      IF finalPosition == 29 THEN
        ;FOLD SPTP P129 Vel=100 % PDAT1 Tool[1]:SMC Base[0] ;%{PE}
        ;FOLD Parameters ;%{h}
        ;Params IlfProvider=kukaroboter.basistech.inlineforms.movement.spline; Kuka.IsGlobalPoint=False; Kuka.PointName=P129; Kuka.BlendingEnabled=False; Kuka.MoveDataPtpName=PDAT1; Kuka.VelocityPtp=100; Kuka.VelocityFieldEnabled=True; Kuka.ColDetectFieldEnabled=True; Kuka.CurrentCDSetIndex=0; Kuka.MovementParameterFieldEnabled=True; IlfCommand=SPTP
        ;ENDFOLD
        SPTP XP129 WITH $VEL_AXIS[1] = SVEL_JOINT(100.0), $TOOL = STOOL2(FP129), $BASE = SBASE(FP129.BASE_NO), $IPO_MODE = SIPO_MODE(FP129.IPO_FRAME), $LOAD = SLOAD(FP129.TOOL_NO), $ACC_AXIS[1] = SACC_JOINT(PPDAT1), $APO = SAPO_PTP(PPDAT1), $GEAR_JERK[1] = SGEAR_JERK(PPDAT1), $COLLMON_TOL_PRO[1] = USE_CM_PRO_VALUES(0)
        ;ENDFOLD
        ;FOLD SLIN P229 Vel=0.1 m/s CPDAT27 Tool[1]:SMC Base[0] ;%{PE}
        ;FOLD Parameters ;%{h}
        ;Params IlfProvider=kukaroboter.basistech.inlineforms.movement.spline; Kuka.IsGlobalPoint=False; Kuka.PointName=P229; Kuka.BlendingEnabled=False; Kuka.MoveDataName=CPDAT27; Kuka.VelocityPath=0.1; Kuka.VelocityFieldEnabled=True; Kuka.ColDetectFieldEnabled=True; Kuka.CurrentCDSetIndex=0; Kuka.MovementParameterFieldEnabled=True; IlfCommand=SLIN
        ;ENDFOLD
        SLIN XP229 WITH $VEL = SVEL_CP(0.1, , LCPDAT27), $TOOL = STOOL2(FP229), $BASE = SBASE(FP229.BASE_NO), $IPO_MODE = SIPO_MODE(FP229.IPO_FRAME), $LOAD = SLOAD(FP229.TOOL_NO), $ACC = SACC_CP(LCPDAT27), $ORI_TYPE = SORI_TYP(LCPDAT27), $APO = SAPO(LCPDAT27), $JERK = SJERK(LCPDAT27), $COLLMON_TOL_PRO[1] = USE_CM_PRO_VALUES(0)
        ;ENDFOLD
        ;FOLD Gripper SET [1]Gripper1 State=[1]ABIERTA Wait 0.2[s] Check with Strategy 1 ;%{PE}
        ;FOLD Parameters Parameters ;%{h}
        ;Params IlfProvider=GripperTech.GripperSet;setgripper=1;setstate=1;setcont=nocont;waittime=0.2;errorstrategy=1
        ;ENDFOLD
        GRPg_SetStateAndCheck(1, 1, 0.2, 1)
        ;ENDFOLD
        ;FOLD SLIN P129 Vel=0.1 m/s CPDAT28 Tool[1]:SMC Base[0] ;%{PE}
        ;FOLD Parameters ;%{h}
        ;Params IlfProvider=kukaroboter.basistech.inlineforms.movement.spline; Kuka.IsGlobalPoint=False; Kuka.PointName=P129; Kuka.BlendingEnabled=False; Kuka.MoveDataName=CPDAT28; Kuka.VelocityPath=0.1; Kuka.VelocityFieldEnabled=True; Kuka.ColDetectFieldEnabled=True; Kuka.CurrentCDSetIndex=0; Kuka.MovementParameterFieldEnabled=True; IlfCommand=SLIN
        ;ENDFOLD
        SLIN XP129 WITH $VEL = SVEL_CP(0.1, , LCPDAT28), $TOOL = STOOL2(FP129), $BASE = SBASE(FP129.BASE_NO), $IPO_MODE = SIPO_MODE(FP129.IPO_FRAME), $LOAD = SLOAD(FP129.TOOL_NO), $ACC = SACC_CP(LCPDAT28), $ORI_TYPE = SORI_TYP(LCPDAT28), $APO = SAPO(LCPDAT28), $JERK = SJERK(LCPDAT28), $COLLMON_TOL_PRO[1] = USE_CM_PRO_VALUES(0)
        ;ENDFOLD
        ;FOLD SPTP P600 Vel=100 % PDAT1 Tool[1]:SMC Base[0] ;%{PE}
        ;FOLD Parameters ;%{h}
        ;Params IlfProvider=kukaroboter.basistech.inlineforms.movement.spline; Kuka.IsGlobalPoint=False; Kuka.PointName=P600; Kuka.BlendingEnabled=False; Kuka.MoveDataPtpName=PDAT1; Kuka.VelocityPtp=100; Kuka.VelocityFieldEnabled=True; Kuka.ColDetectFieldEnabled=True; Kuka.CurrentCDSetIndex=0; Kuka.MovementParameterFieldEnabled=True; IlfCommand=SPTP
        ;ENDFOLD
        SPTP XP600 WITH $VEL_AXIS[1] = SVEL_JOINT(100.0), $TOOL = STOOL2(FP600), $BASE = SBASE(FP600.BASE_NO), $IPO_MODE = SIPO_MODE(FP600.IPO_FRAME), $LOAD = SLOAD(FP600.TOOL_NO), $ACC_AXIS[1] = SACC_JOINT(PPDAT1), $APO = SAPO_PTP(PPDAT1), $GEAR_JERK[1] = SGEAR_JERK(PPDAT1), $COLLMON_TOL_PRO[1] = USE_CM_PRO_VALUES(0)
        ;ENDFOLD
        ;FOLD SLIN P601 Vel=0.1 m/s CPDAT27 Tool[1]:SMC Base[0] ;%{PE}
        ;FOLD Parameters ;%{h}
        ;Params IlfProvider=kukaroboter.basistech.inlineforms.movement.spline; Kuka.IsGlobalPoint=False; Kuka.PointName=P601; Kuka.BlendingEnabled=False; Kuka.MoveDataName=CPDAT27; Kuka.VelocityPath=0.1; Kuka.VelocityFieldEnabled=True; Kuka.ColDetectFieldEnabled=True; Kuka.CurrentCDSetIndex=0; Kuka.MovementParameterFieldEnabled=True; IlfCommand=SLIN
        ;ENDFOLD
        SLIN XP601 WITH $VEL = SVEL_CP(0.1, , LCPDAT27), $TOOL = STOOL2(FP601), $BASE = SBASE(FP601.BASE_NO), $IPO_MODE = SIPO_MODE(FP601.IPO_FRAME), $LOAD = SLOAD(FP601.TOOL_NO), $ACC = SACC_CP(LCPDAT27), $ORI_TYPE = SORI_TYP(LCPDAT27), $APO = SAPO(LCPDAT27), $JERK = SJERK(LCPDAT27), $COLLMON_TOL_PRO[1] = USE_CM_PRO_VALUES(0)
        ;ENDFOLD
        ;FOLD SLIN P602 Vel=0.1 m/s CPDAT27 Tool[1]:SMC Base[0] ;%{PE}
        ;FOLD Parameters ;%{h}
        ;Params IlfProvider=kukaroboter.basistech.inlineforms.movement.spline; Kuka.IsGlobalPoint=False; Kuka.PointName=P602; Kuka.BlendingEnabled=False; Kuka.MoveDataName=CPDAT27; Kuka.VelocityPath=0.1; Kuka.VelocityFieldEnabled=True; Kuka.ColDetectFieldEnabled=True; Kuka.CurrentCDSetIndex=0; Kuka.MovementParameterFieldEnabled=True; IlfCommand=SLIN
        ;ENDFOLD
        SLIN XP602 WITH $VEL = SVEL_CP(0.1, , LCPDAT27), $TOOL = STOOL2(FP602), $BASE = SBASE(FP602.BASE_NO), $IPO_MODE = SIPO_MODE(FP602.IPO_FRAME), $LOAD = SLOAD(FP602.TOOL_NO), $ACC = SACC_CP(LCPDAT27), $ORI_TYPE = SORI_TYP(LCPDAT27), $APO = SAPO(LCPDAT27), $JERK = SJERK(LCPDAT27), $COLLMON_TOL_PRO[1] = USE_CM_PRO_VALUES(0)
        ;ENDFOLD
      ENDIF

      IF finalPosition == 30 THEN
        ;FOLD SPTP P130 Vel=100 % PDAT1 Tool[1]:SMC Base[0] ;%{PE}
        ;FOLD Parameters ;%{h}
        ;Params IlfProvider=kukaroboter.basistech.inlineforms.movement.spline; Kuka.IsGlobalPoint=False; Kuka.PointName=P130; Kuka.BlendingEnabled=False; Kuka.MoveDataPtpName=PDAT1; Kuka.VelocityPtp=100; Kuka.VelocityFieldEnabled=True; Kuka.ColDetectFieldEnabled=True; Kuka.CurrentCDSetIndex=0; Kuka.MovementParameterFieldEnabled=True; IlfCommand=SPTP
        ;ENDFOLD
        SPTP XP130 WITH $VEL_AXIS[1] = SVEL_JOINT(100.0), $TOOL = STOOL2(FP130), $BASE = SBASE(FP130.BASE_NO), $IPO_MODE = SIPO_MODE(FP130.IPO_FRAME), $LOAD = SLOAD(FP130.TOOL_NO), $ACC_AXIS[1] = SACC_JOINT(PPDAT1), $APO = SAPO_PTP(PPDAT1), $GEAR_JERK[1] = SGEAR_JERK(PPDAT1), $COLLMON_TOL_PRO[1] = USE_CM_PRO_VALUES(0)
        ;ENDFOLD
        ;FOLD SLIN P230 Vel=0.1 m/s CPDAT27 Tool[1]:SMC Base[0] ;%{PE}
        ;FOLD Parameters ;%{h}
        ;Params IlfProvider=kukaroboter.basistech.inlineforms.movement.spline; Kuka.IsGlobalPoint=False; Kuka.PointName=P230; Kuka.BlendingEnabled=False; Kuka.MoveDataName=CPDAT27; Kuka.VelocityPath=0.1; Kuka.VelocityFieldEnabled=True; Kuka.ColDetectFieldEnabled=True; Kuka.CurrentCDSetIndex=0; Kuka.MovementParameterFieldEnabled=True; IlfCommand=SLIN
        ;ENDFOLD
        SLIN XP230 WITH $VEL = SVEL_CP(0.1, , LCPDAT27), $TOOL = STOOL2(FP230), $BASE = SBASE(FP230.BASE_NO), $IPO_MODE = SIPO_MODE(FP230.IPO_FRAME), $LOAD = SLOAD(FP230.TOOL_NO), $ACC = SACC_CP(LCPDAT27), $ORI_TYPE = SORI_TYP(LCPDAT27), $APO = SAPO(LCPDAT27), $JERK = SJERK(LCPDAT27), $COLLMON_TOL_PRO[1] = USE_CM_PRO_VALUES(0)
        ;ENDFOLD
        ;FOLD Gripper SET [1]Gripper1 State=[1]ABIERTA Wait 0.2[s] Check with Strategy 1 ;%{PE}
        ;FOLD Parameters Parameters ;%{h}
        ;Params IlfProvider=GripperTech.GripperSet;setgripper=1;setstate=1;setcont=nocont;waittime=0.2;errorstrategy=1
        ;ENDFOLD
        GRPg_SetStateAndCheck(1, 1, 0.2, 1)
        ;ENDFOLD
        ;FOLD SLIN P130 Vel=0.1 m/s CPDAT28 Tool[1]:SMC Base[0] ;%{PE}
        ;FOLD Parameters ;%{h}
        ;Params IlfProvider=kukaroboter.basistech.inlineforms.movement.spline; Kuka.IsGlobalPoint=False; Kuka.PointName=P130; Kuka.BlendingEnabled=False; Kuka.MoveDataName=CPDAT28; Kuka.VelocityPath=0.1; Kuka.VelocityFieldEnabled=True; Kuka.ColDetectFieldEnabled=True; Kuka.CurrentCDSetIndex=0; Kuka.MovementParameterFieldEnabled=True; IlfCommand=SLIN
        ;ENDFOLD
        SLIN XP130 WITH $VEL = SVEL_CP(0.1, , LCPDAT28), $TOOL = STOOL2(FP130), $BASE = SBASE(FP130.BASE_NO), $IPO_MODE = SIPO_MODE(FP130.IPO_FRAME), $LOAD = SLOAD(FP130.TOOL_NO), $ACC = SACC_CP(LCPDAT28), $ORI_TYPE = SORI_TYP(LCPDAT28), $APO = SAPO(LCPDAT28), $JERK = SJERK(LCPDAT28), $COLLMON_TOL_PRO[1] = USE_CM_PRO_VALUES(0)
        ;ENDFOLD
        ;FOLD SPTP P600 Vel=100 % PDAT1 Tool[1]:SMC Base[0] ;%{PE}
        ;FOLD Parameters ;%{h}
        ;Params IlfProvider=kukaroboter.basistech.inlineforms.movement.spline; Kuka.IsGlobalPoint=False; Kuka.PointName=P600; Kuka.BlendingEnabled=False; Kuka.MoveDataPtpName=PDAT1; Kuka.VelocityPtp=100; Kuka.VelocityFieldEnabled=True; Kuka.ColDetectFieldEnabled=True; Kuka.CurrentCDSetIndex=0; Kuka.MovementParameterFieldEnabled=True; IlfCommand=SPTP
        ;ENDFOLD
        SPTP XP600 WITH $VEL_AXIS[1] = SVEL_JOINT(100.0), $TOOL = STOOL2(FP600), $BASE = SBASE(FP600.BASE_NO), $IPO_MODE = SIPO_MODE(FP600.IPO_FRAME), $LOAD = SLOAD(FP600.TOOL_NO), $ACC_AXIS[1] = SACC_JOINT(PPDAT1), $APO = SAPO_PTP(PPDAT1), $GEAR_JERK[1] = SGEAR_JERK(PPDAT1), $COLLMON_TOL_PRO[1] = USE_CM_PRO_VALUES(0)
        ;ENDFOLD
        ;FOLD SLIN P601 Vel=0.1 m/s CPDAT27 Tool[1]:SMC Base[0] ;%{PE}
        ;FOLD Parameters ;%{h}
        ;Params IlfProvider=kukaroboter.basistech.inlineforms.movement.spline; Kuka.IsGlobalPoint=False; Kuka.PointName=P601; Kuka.BlendingEnabled=False; Kuka.MoveDataName=CPDAT27; Kuka.VelocityPath=0.1; Kuka.VelocityFieldEnabled=True; Kuka.ColDetectFieldEnabled=True; Kuka.CurrentCDSetIndex=0; Kuka.MovementParameterFieldEnabled=True; IlfCommand=SLIN
        ;ENDFOLD
        SLIN XP601 WITH $VEL = SVEL_CP(0.1, , LCPDAT27), $TOOL = STOOL2(FP601), $BASE = SBASE(FP601.BASE_NO), $IPO_MODE = SIPO_MODE(FP601.IPO_FRAME), $LOAD = SLOAD(FP601.TOOL_NO), $ACC = SACC_CP(LCPDAT27), $ORI_TYPE = SORI_TYP(LCPDAT27), $APO = SAPO(LCPDAT27), $JERK = SJERK(LCPDAT27), $COLLMON_TOL_PRO[1] = USE_CM_PRO_VALUES(0)
        ;ENDFOLD
        ;FOLD SLIN P602 Vel=0.1 m/s CPDAT27 Tool[1]:SMC Base[0] ;%{PE}
        ;FOLD Parameters ;%{h}
        ;Params IlfProvider=kukaroboter.basistech.inlineforms.movement.spline; Kuka.IsGlobalPoint=False; Kuka.PointName=P602; Kuka.BlendingEnabled=False; Kuka.MoveDataName=CPDAT27; Kuka.VelocityPath=0.1; Kuka.VelocityFieldEnabled=True; Kuka.ColDetectFieldEnabled=True; Kuka.CurrentCDSetIndex=0; Kuka.MovementParameterFieldEnabled=True; IlfCommand=SLIN
        ;ENDFOLD
        SLIN XP602 WITH $VEL = SVEL_CP(0.1, , LCPDAT27), $TOOL = STOOL2(FP602), $BASE = SBASE(FP602.BASE_NO), $IPO_MODE = SIPO_MODE(FP602.IPO_FRAME), $LOAD = SLOAD(FP602.TOOL_NO), $ACC = SACC_CP(LCPDAT27), $ORI_TYPE = SORI_TYP(LCPDAT27), $APO = SAPO(LCPDAT27), $JERK = SJERK(LCPDAT27), $COLLMON_TOL_PRO[1] = USE_CM_PRO_VALUES(0)
        ;ENDFOLD
      ENDIF

      IF finalPosition == 31 THEN
        ;FOLD SPTP P131 Vel=100 % PDAT1 Tool[1]:SMC Base[0] ;%{PE}
        ;FOLD Parameters ;%{h}
        ;Params IlfProvider=kukaroboter.basistech.inlineforms.movement.spline; Kuka.IsGlobalPoint=False; Kuka.PointName=P131; Kuka.BlendingEnabled=False; Kuka.MoveDataPtpName=PDAT1; Kuka.VelocityPtp=100; Kuka.VelocityFieldEnabled=True; Kuka.ColDetectFieldEnabled=True; Kuka.CurrentCDSetIndex=0; Kuka.MovementParameterFieldEnabled=True; IlfCommand=SPTP
        ;ENDFOLD
        SPTP XP131 WITH $VEL_AXIS[1] = SVEL_JOINT(100.0), $TOOL = STOOL2(FP131), $BASE = SBASE(FP131.BASE_NO), $IPO_MODE = SIPO_MODE(FP131.IPO_FRAME), $LOAD = SLOAD(FP131.TOOL_NO), $ACC_AXIS[1] = SACC_JOINT(PPDAT1), $APO = SAPO_PTP(PPDAT1), $GEAR_JERK[1] = SGEAR_JERK(PPDAT1), $COLLMON_TOL_PRO[1] = USE_CM_PRO_VALUES(0)
        ;ENDFOLD
        ;FOLD SLIN P231 Vel=0.1 m/s CPDAT27 Tool[1]:SMC Base[0] ;%{PE}
        ;FOLD Parameters ;%{h}
        ;Params IlfProvider=kukaroboter.basistech.inlineforms.movement.spline; Kuka.IsGlobalPoint=False; Kuka.PointName=P231; Kuka.BlendingEnabled=False; Kuka.MoveDataName=CPDAT27; Kuka.VelocityPath=0.1; Kuka.VelocityFieldEnabled=True; Kuka.ColDetectFieldEnabled=True; Kuka.CurrentCDSetIndex=0; Kuka.MovementParameterFieldEnabled=True; IlfCommand=SLIN
        ;ENDFOLD
        SLIN XP231 WITH $VEL = SVEL_CP(0.1, , LCPDAT27), $TOOL = STOOL2(FP231), $BASE = SBASE(FP231.BASE_NO), $IPO_MODE = SIPO_MODE(FP231.IPO_FRAME), $LOAD = SLOAD(FP231.TOOL_NO), $ACC = SACC_CP(LCPDAT27), $ORI_TYPE = SORI_TYP(LCPDAT27), $APO = SAPO(LCPDAT27), $JERK = SJERK(LCPDAT27), $COLLMON_TOL_PRO[1] = USE_CM_PRO_VALUES(0)
        ;ENDFOLD
        ;FOLD Gripper SET [1]Gripper1 State=[1]ABIERTA Wait 0.2[s] Check with Strategy 1 ;%{PE}
        ;FOLD Parameters Parameters ;%{h}
        ;Params IlfProvider=GripperTech.GripperSet;setgripper=1;setstate=1;setcont=nocont;waittime=0.2;errorstrategy=1
        ;ENDFOLD
        GRPg_SetStateAndCheck(1, 1, 0.2, 1)
        ;ENDFOLD
        ;FOLD SLIN P131 Vel=0.1 m/s CPDAT28 Tool[1]:SMC Base[0] ;%{PE}
        ;FOLD Parameters ;%{h}
        ;Params IlfProvider=kukaroboter.basistech.inlineforms.movement.spline; Kuka.IsGlobalPoint=False; Kuka.PointName=P131; Kuka.BlendingEnabled=False; Kuka.MoveDataName=CPDAT28; Kuka.VelocityPath=0.1; Kuka.VelocityFieldEnabled=True; Kuka.ColDetectFieldEnabled=True; Kuka.CurrentCDSetIndex=0; Kuka.MovementParameterFieldEnabled=True; IlfCommand=SLIN
        ;ENDFOLD
        SLIN XP131 WITH $VEL = SVEL_CP(0.1, , LCPDAT28), $TOOL = STOOL2(FP131), $BASE = SBASE(FP131.BASE_NO), $IPO_MODE = SIPO_MODE(FP131.IPO_FRAME), $LOAD = SLOAD(FP131.TOOL_NO), $ACC = SACC_CP(LCPDAT28), $ORI_TYPE = SORI_TYP(LCPDAT28), $APO = SAPO(LCPDAT28), $JERK = SJERK(LCPDAT28), $COLLMON_TOL_PRO[1] = USE_CM_PRO_VALUES(0)
        ;ENDFOLD
        ;FOLD SPTP P600 Vel=100 % PDAT1 Tool[1]:SMC Base[0] ;%{PE}
        ;FOLD Parameters ;%{h}
        ;Params IlfProvider=kukaroboter.basistech.inlineforms.movement.spline; Kuka.IsGlobalPoint=False; Kuka.PointName=P600; Kuka.BlendingEnabled=False; Kuka.MoveDataPtpName=PDAT1; Kuka.VelocityPtp=100; Kuka.VelocityFieldEnabled=True; Kuka.ColDetectFieldEnabled=True; Kuka.CurrentCDSetIndex=0; Kuka.MovementParameterFieldEnabled=True; IlfCommand=SPTP
        ;ENDFOLD
        SPTP XP600 WITH $VEL_AXIS[1] = SVEL_JOINT(100.0), $TOOL = STOOL2(FP600), $BASE = SBASE(FP600.BASE_NO), $IPO_MODE = SIPO_MODE(FP600.IPO_FRAME), $LOAD = SLOAD(FP600.TOOL_NO), $ACC_AXIS[1] = SACC_JOINT(PPDAT1), $APO = SAPO_PTP(PPDAT1), $GEAR_JERK[1] = SGEAR_JERK(PPDAT1), $COLLMON_TOL_PRO[1] = USE_CM_PRO_VALUES(0)
        ;ENDFOLD
        ;FOLD SLIN P601 Vel=0.1 m/s CPDAT27 Tool[1]:SMC Base[0] ;%{PE}
        ;FOLD Parameters ;%{h}
        ;Params IlfProvider=kukaroboter.basistech.inlineforms.movement.spline; Kuka.IsGlobalPoint=False; Kuka.PointName=P601; Kuka.BlendingEnabled=False; Kuka.MoveDataName=CPDAT27; Kuka.VelocityPath=0.1; Kuka.VelocityFieldEnabled=True; Kuka.ColDetectFieldEnabled=True; Kuka.CurrentCDSetIndex=0; Kuka.MovementParameterFieldEnabled=True; IlfCommand=SLIN
        ;ENDFOLD
        SLIN XP601 WITH $VEL = SVEL_CP(0.1, , LCPDAT27), $TOOL = STOOL2(FP601), $BASE = SBASE(FP601.BASE_NO), $IPO_MODE = SIPO_MODE(FP601.IPO_FRAME), $LOAD = SLOAD(FP601.TOOL_NO), $ACC = SACC_CP(LCPDAT27), $ORI_TYPE = SORI_TYP(LCPDAT27), $APO = SAPO(LCPDAT27), $JERK = SJERK(LCPDAT27), $COLLMON_TOL_PRO[1] = USE_CM_PRO_VALUES(0)
        ;ENDFOLD
        ;FOLD SLIN P602 Vel=0.1 m/s CPDAT27 Tool[1]:SMC Base[0] ;%{PE}
        ;FOLD Parameters ;%{h}
        ;Params IlfProvider=kukaroboter.basistech.inlineforms.movement.spline; Kuka.IsGlobalPoint=False; Kuka.PointName=P602; Kuka.BlendingEnabled=False; Kuka.MoveDataName=CPDAT27; Kuka.VelocityPath=0.1; Kuka.VelocityFieldEnabled=True; Kuka.ColDetectFieldEnabled=True; Kuka.CurrentCDSetIndex=0; Kuka.MovementParameterFieldEnabled=True; IlfCommand=SLIN
        ;ENDFOLD
        SLIN XP602 WITH $VEL = SVEL_CP(0.1, , LCPDAT27), $TOOL = STOOL2(FP602), $BASE = SBASE(FP602.BASE_NO), $IPO_MODE = SIPO_MODE(FP602.IPO_FRAME), $LOAD = SLOAD(FP602.TOOL_NO), $ACC = SACC_CP(LCPDAT27), $ORI_TYPE = SORI_TYP(LCPDAT27), $APO = SAPO(LCPDAT27), $JERK = SJERK(LCPDAT27), $COLLMON_TOL_PRO[1] = USE_CM_PRO_VALUES(0)
        ;ENDFOLD
      ENDIF

      IF finalPosition == 32 THEN
        ;FOLD SPTP P132 Vel=100 % PDAT1 Tool[1]:SMC Base[0] ;%{PE}
        ;FOLD Parameters ;%{h}
        ;Params IlfProvider=kukaroboter.basistech.inlineforms.movement.spline; Kuka.IsGlobalPoint=False; Kuka.PointName=P132; Kuka.BlendingEnabled=False; Kuka.MoveDataPtpName=PDAT1; Kuka.VelocityPtp=100; Kuka.VelocityFieldEnabled=True; Kuka.ColDetectFieldEnabled=True; Kuka.CurrentCDSetIndex=0; Kuka.MovementParameterFieldEnabled=True; IlfCommand=SPTP
        ;ENDFOLD
        SPTP XP132 WITH $VEL_AXIS[1] = SVEL_JOINT(100.0), $TOOL = STOOL2(FP132), $BASE = SBASE(FP132.BASE_NO), $IPO_MODE = SIPO_MODE(FP132.IPO_FRAME), $LOAD = SLOAD(FP132.TOOL_NO), $ACC_AXIS[1] = SACC_JOINT(PPDAT1), $APO = SAPO_PTP(PPDAT1), $GEAR_JERK[1] = SGEAR_JERK(PPDAT1), $COLLMON_TOL_PRO[1] = USE_CM_PRO_VALUES(0)
        ;ENDFOLD
        ;FOLD SLIN P232 Vel=0.1 m/s CPDAT27 Tool[1]:SMC Base[0] ;%{PE}
        ;FOLD Parameters ;%{h}
        ;Params IlfProvider=kukaroboter.basistech.inlineforms.movement.spline; Kuka.IsGlobalPoint=False; Kuka.PointName=P232; Kuka.BlendingEnabled=False; Kuka.MoveDataName=CPDAT27; Kuka.VelocityPath=0.1; Kuka.VelocityFieldEnabled=True; Kuka.ColDetectFieldEnabled=True; Kuka.CurrentCDSetIndex=0; Kuka.MovementParameterFieldEnabled=True; IlfCommand=SLIN
        ;ENDFOLD
        SLIN XP232 WITH $VEL = SVEL_CP(0.1, , LCPDAT27), $TOOL = STOOL2(FP232), $BASE = SBASE(FP232.BASE_NO), $IPO_MODE = SIPO_MODE(FP232.IPO_FRAME), $LOAD = SLOAD(FP232.TOOL_NO), $ACC = SACC_CP(LCPDAT27), $ORI_TYPE = SORI_TYP(LCPDAT27), $APO = SAPO(LCPDAT27), $JERK = SJERK(LCPDAT27), $COLLMON_TOL_PRO[1] = USE_CM_PRO_VALUES(0)
        ;ENDFOLD
        ;FOLD Gripper SET [1]Gripper1 State=[1]ABIERTA Wait 0.2[s] Check with Strategy 1 ;%{PE}
        ;FOLD Parameters Parameters ;%{h}
        ;Params IlfProvider=GripperTech.GripperSet;setgripper=1;setstate=1;setcont=nocont;waittime=0.2;errorstrategy=1
        ;ENDFOLD
        GRPg_SetStateAndCheck(1, 1, 0.2, 1)
        ;ENDFOLD
        ;FOLD SLIN P132 Vel=0.1 m/s CPDAT28 Tool[1]:SMC Base[0] ;%{PE}
        ;FOLD Parameters ;%{h}
        ;Params IlfProvider=kukaroboter.basistech.inlineforms.movement.spline; Kuka.IsGlobalPoint=False; Kuka.PointName=P132; Kuka.BlendingEnabled=False; Kuka.MoveDataName=CPDAT28; Kuka.VelocityPath=0.1; Kuka.VelocityFieldEnabled=True; Kuka.ColDetectFieldEnabled=True; Kuka.CurrentCDSetIndex=0; Kuka.MovementParameterFieldEnabled=True; IlfCommand=SLIN
        ;ENDFOLD
        SLIN XP132 WITH $VEL = SVEL_CP(0.1, , LCPDAT28), $TOOL = STOOL2(FP132), $BASE = SBASE(FP132.BASE_NO), $IPO_MODE = SIPO_MODE(FP132.IPO_FRAME), $LOAD = SLOAD(FP132.TOOL_NO), $ACC = SACC_CP(LCPDAT28), $ORI_TYPE = SORI_TYP(LCPDAT28), $APO = SAPO(LCPDAT28), $JERK = SJERK(LCPDAT28), $COLLMON_TOL_PRO[1] = USE_CM_PRO_VALUES(0)
        ;ENDFOLD
        ;FOLD SPTP P600 Vel=100 % PDAT1 Tool[1]:SMC Base[0] ;%{PE}
        ;FOLD Parameters ;%{h}
        ;Params IlfProvider=kukaroboter.basistech.inlineforms.movement.spline; Kuka.IsGlobalPoint=False; Kuka.PointName=P600; Kuka.BlendingEnabled=False; Kuka.MoveDataPtpName=PDAT1; Kuka.VelocityPtp=100; Kuka.VelocityFieldEnabled=True; Kuka.ColDetectFieldEnabled=True; Kuka.CurrentCDSetIndex=0; Kuka.MovementParameterFieldEnabled=True; IlfCommand=SPTP
        ;ENDFOLD
        SPTP XP600 WITH $VEL_AXIS[1] = SVEL_JOINT(100.0), $TOOL = STOOL2(FP600), $BASE = SBASE(FP600.BASE_NO), $IPO_MODE = SIPO_MODE(FP600.IPO_FRAME), $LOAD = SLOAD(FP600.TOOL_NO), $ACC_AXIS[1] = SACC_JOINT(PPDAT1), $APO = SAPO_PTP(PPDAT1), $GEAR_JERK[1] = SGEAR_JERK(PPDAT1), $COLLMON_TOL_PRO[1] = USE_CM_PRO_VALUES(0)
        ;ENDFOLD
        ;FOLD SLIN P601 Vel=0.1 m/s CPDAT27 Tool[1]:SMC Base[0] ;%{PE}
        ;FOLD Parameters ;%{h}
        ;Params IlfProvider=kukaroboter.basistech.inlineforms.movement.spline; Kuka.IsGlobalPoint=False; Kuka.PointName=P601; Kuka.BlendingEnabled=False; Kuka.MoveDataName=CPDAT27; Kuka.VelocityPath=0.1; Kuka.VelocityFieldEnabled=True; Kuka.ColDetectFieldEnabled=True; Kuka.CurrentCDSetIndex=0; Kuka.MovementParameterFieldEnabled=True; IlfCommand=SLIN
        ;ENDFOLD
        SLIN XP601 WITH $VEL = SVEL_CP(0.1, , LCPDAT27), $TOOL = STOOL2(FP601), $BASE = SBASE(FP601.BASE_NO), $IPO_MODE = SIPO_MODE(FP601.IPO_FRAME), $LOAD = SLOAD(FP601.TOOL_NO), $ACC = SACC_CP(LCPDAT27), $ORI_TYPE = SORI_TYP(LCPDAT27), $APO = SAPO(LCPDAT27), $JERK = SJERK(LCPDAT27), $COLLMON_TOL_PRO[1] = USE_CM_PRO_VALUES(0)
        ;ENDFOLD
        ;FOLD SLIN P602 Vel=0.1 m/s CPDAT27 Tool[1]:SMC Base[0] ;%{PE}
        ;FOLD Parameters ;%{h}
        ;Params IlfProvider=kukaroboter.basistech.inlineforms.movement.spline; Kuka.IsGlobalPoint=False; Kuka.PointName=P602; Kuka.BlendingEnabled=False; Kuka.MoveDataName=CPDAT27; Kuka.VelocityPath=0.1; Kuka.VelocityFieldEnabled=True; Kuka.ColDetectFieldEnabled=True; Kuka.CurrentCDSetIndex=0; Kuka.MovementParameterFieldEnabled=True; IlfCommand=SLIN
        ;ENDFOLD
        SLIN XP602 WITH $VEL = SVEL_CP(0.1, , LCPDAT27), $TOOL = STOOL2(FP602), $BASE = SBASE(FP602.BASE_NO), $IPO_MODE = SIPO_MODE(FP602.IPO_FRAME), $LOAD = SLOAD(FP602.TOOL_NO), $ACC = SACC_CP(LCPDAT27), $ORI_TYPE = SORI_TYP(LCPDAT27), $APO = SAPO(LCPDAT27), $JERK = SJERK(LCPDAT27), $COLLMON_TOL_PRO[1] = USE_CM_PRO_VALUES(0)
        ;ENDFOLD
      ENDIF

      IF finalPosition == 33 THEN
        ;FOLD SPTP P133 Vel=100 % PDAT1 Tool[1]:SMC Base[0] ;%{PE}
        ;FOLD Parameters ;%{h}
        ;Params IlfProvider=kukaroboter.basistech.inlineforms.movement.spline; Kuka.IsGlobalPoint=False; Kuka.PointName=P133; Kuka.BlendingEnabled=False; Kuka.MoveDataPtpName=PDAT1; Kuka.VelocityPtp=100; Kuka.VelocityFieldEnabled=True; Kuka.ColDetectFieldEnabled=True; Kuka.CurrentCDSetIndex=0; Kuka.MovementParameterFieldEnabled=True; IlfCommand=SPTP
        ;ENDFOLD
        SPTP XP133 WITH $VEL_AXIS[1] = SVEL_JOINT(100.0), $TOOL = STOOL2(FP133), $BASE = SBASE(FP133.BASE_NO), $IPO_MODE = SIPO_MODE(FP133.IPO_FRAME), $LOAD = SLOAD(FP133.TOOL_NO), $ACC_AXIS[1] = SACC_JOINT(PPDAT1), $APO = SAPO_PTP(PPDAT1), $GEAR_JERK[1] = SGEAR_JERK(PPDAT1), $COLLMON_TOL_PRO[1] = USE_CM_PRO_VALUES(0)
        ;ENDFOLD
        ;FOLD SLIN P233 Vel=0.1 m/s CPDAT27 Tool[1]:SMC Base[0] ;%{PE}
        ;FOLD Parameters ;%{h}
        ;Params IlfProvider=kukaroboter.basistech.inlineforms.movement.spline; Kuka.IsGlobalPoint=False; Kuka.PointName=P233; Kuka.BlendingEnabled=False; Kuka.MoveDataName=CPDAT27; Kuka.VelocityPath=0.1; Kuka.VelocityFieldEnabled=True; Kuka.ColDetectFieldEnabled=True; Kuka.CurrentCDSetIndex=0; Kuka.MovementParameterFieldEnabled=True; IlfCommand=SLIN
        ;ENDFOLD
        SLIN XP233 WITH $VEL = SVEL_CP(0.1, , LCPDAT27), $TOOL = STOOL2(FP233), $BASE = SBASE(FP233.BASE_NO), $IPO_MODE = SIPO_MODE(FP233.IPO_FRAME), $LOAD = SLOAD(FP233.TOOL_NO), $ACC = SACC_CP(LCPDAT27), $ORI_TYPE = SORI_TYP(LCPDAT27), $APO = SAPO(LCPDAT27), $JERK = SJERK(LCPDAT27), $COLLMON_TOL_PRO[1] = USE_CM_PRO_VALUES(0)
        ;ENDFOLD
        ;FOLD Gripper SET [1]Gripper1 State=[1]ABIERTA Wait 0.2[s] Check with Strategy 1 ;%{PE}
        ;FOLD Parameters Parameters ;%{h}
        ;Params IlfProvider=GripperTech.GripperSet;setgripper=1;setstate=1;setcont=nocont;waittime=0.2;errorstrategy=1
        ;ENDFOLD
        GRPg_SetStateAndCheck(1, 1, 0.2, 1)
        ;ENDFOLD
        ;FOLD SLIN P133 Vel=0.1 m/s CPDAT28 Tool[1]:SMC Base[0] ;%{PE}
        ;FOLD Parameters ;%{h}
        ;Params IlfProvider=kukaroboter.basistech.inlineforms.movement.spline; Kuka.IsGlobalPoint=False; Kuka.PointName=P133; Kuka.BlendingEnabled=False; Kuka.MoveDataName=CPDAT28; Kuka.VelocityPath=0.1; Kuka.VelocityFieldEnabled=True; Kuka.ColDetectFieldEnabled=True; Kuka.CurrentCDSetIndex=0; Kuka.MovementParameterFieldEnabled=True; IlfCommand=SLIN
        ;ENDFOLD
        SLIN XP133 WITH $VEL = SVEL_CP(0.1, , LCPDAT28), $TOOL = STOOL2(FP133), $BASE = SBASE(FP133.BASE_NO), $IPO_MODE = SIPO_MODE(FP133.IPO_FRAME), $LOAD = SLOAD(FP133.TOOL_NO), $ACC = SACC_CP(LCPDAT28), $ORI_TYPE = SORI_TYP(LCPDAT28), $APO = SAPO(LCPDAT28), $JERK = SJERK(LCPDAT28), $COLLMON_TOL_PRO[1] = USE_CM_PRO_VALUES(0)
        ;ENDFOLD
        ;FOLD SPTP P600 Vel=100 % PDAT1 Tool[1]:SMC Base[0] ;%{PE}
        ;FOLD Parameters ;%{h}
        ;Params IlfProvider=kukaroboter.basistech.inlineforms.movement.spline; Kuka.IsGlobalPoint=False; Kuka.PointName=P600; Kuka.BlendingEnabled=False; Kuka.MoveDataPtpName=PDAT1; Kuka.VelocityPtp=100; Kuka.VelocityFieldEnabled=True; Kuka.ColDetectFieldEnabled=True; Kuka.CurrentCDSetIndex=0; Kuka.MovementParameterFieldEnabled=True; IlfCommand=SPTP
        ;ENDFOLD
        SPTP XP600 WITH $VEL_AXIS[1] = SVEL_JOINT(100.0), $TOOL = STOOL2(FP600), $BASE = SBASE(FP600.BASE_NO), $IPO_MODE = SIPO_MODE(FP600.IPO_FRAME), $LOAD = SLOAD(FP600.TOOL_NO), $ACC_AXIS[1] = SACC_JOINT(PPDAT1), $APO = SAPO_PTP(PPDAT1), $GEAR_JERK[1] = SGEAR_JERK(PPDAT1), $COLLMON_TOL_PRO[1] = USE_CM_PRO_VALUES(0)
        ;ENDFOLD
        ;FOLD SLIN P601 Vel=0.1 m/s CPDAT27 Tool[1]:SMC Base[0] ;%{PE}
        ;FOLD Parameters ;%{h}
        ;Params IlfProvider=kukaroboter.basistech.inlineforms.movement.spline; Kuka.IsGlobalPoint=False; Kuka.PointName=P601; Kuka.BlendingEnabled=False; Kuka.MoveDataName=CPDAT27; Kuka.VelocityPath=0.1; Kuka.VelocityFieldEnabled=True; Kuka.ColDetectFieldEnabled=True; Kuka.CurrentCDSetIndex=0; Kuka.MovementParameterFieldEnabled=True; IlfCommand=SLIN
        ;ENDFOLD
        SLIN XP601 WITH $VEL = SVEL_CP(0.1, , LCPDAT27), $TOOL = STOOL2(FP601), $BASE = SBASE(FP601.BASE_NO), $IPO_MODE = SIPO_MODE(FP601.IPO_FRAME), $LOAD = SLOAD(FP601.TOOL_NO), $ACC = SACC_CP(LCPDAT27), $ORI_TYPE = SORI_TYP(LCPDAT27), $APO = SAPO(LCPDAT27), $JERK = SJERK(LCPDAT27), $COLLMON_TOL_PRO[1] = USE_CM_PRO_VALUES(0)
        ;ENDFOLD
        ;FOLD SLIN P602 Vel=0.1 m/s CPDAT27 Tool[1]:SMC Base[0] ;%{PE}
        ;FOLD Parameters ;%{h}
        ;Params IlfProvider=kukaroboter.basistech.inlineforms.movement.spline; Kuka.IsGlobalPoint=False; Kuka.PointName=P602; Kuka.BlendingEnabled=False; Kuka.MoveDataName=CPDAT27; Kuka.VelocityPath=0.1; Kuka.VelocityFieldEnabled=True; Kuka.ColDetectFieldEnabled=True; Kuka.CurrentCDSetIndex=0; Kuka.MovementParameterFieldEnabled=True; IlfCommand=SLIN
        ;ENDFOLD
        SLIN XP602 WITH $VEL = SVEL_CP(0.1, , LCPDAT27), $TOOL = STOOL2(FP602), $BASE = SBASE(FP602.BASE_NO), $IPO_MODE = SIPO_MODE(FP602.IPO_FRAME), $LOAD = SLOAD(FP602.TOOL_NO), $ACC = SACC_CP(LCPDAT27), $ORI_TYPE = SORI_TYP(LCPDAT27), $APO = SAPO(LCPDAT27), $JERK = SJERK(LCPDAT27), $COLLMON_TOL_PRO[1] = USE_CM_PRO_VALUES(0)
        ;ENDFOLD
      ENDIF

      IF finalPosition == 34 THEN
        ;FOLD SPTP P134 Vel=100 % PDAT1 Tool[1]:SMC Base[0] ;%{PE}
        ;FOLD Parameters ;%{h}
        ;Params IlfProvider=kukaroboter.basistech.inlineforms.movement.spline; Kuka.IsGlobalPoint=False; Kuka.PointName=P134; Kuka.BlendingEnabled=False; Kuka.MoveDataPtpName=PDAT1; Kuka.VelocityPtp=100; Kuka.VelocityFieldEnabled=True; Kuka.ColDetectFieldEnabled=True; Kuka.CurrentCDSetIndex=0; Kuka.MovementParameterFieldEnabled=True; IlfCommand=SPTP
        ;ENDFOLD
        SPTP XP134 WITH $VEL_AXIS[1] = SVEL_JOINT(100.0), $TOOL = STOOL2(FP134), $BASE = SBASE(FP134.BASE_NO), $IPO_MODE = SIPO_MODE(FP134.IPO_FRAME), $LOAD = SLOAD(FP134.TOOL_NO), $ACC_AXIS[1] = SACC_JOINT(PPDAT1), $APO = SAPO_PTP(PPDAT1), $GEAR_JERK[1] = SGEAR_JERK(PPDAT1), $COLLMON_TOL_PRO[1] = USE_CM_PRO_VALUES(0)
        ;ENDFOLD
        ;FOLD SLIN P234 Vel=0.1 m/s CPDAT27 Tool[1]:SMC Base[0] ;%{PE}
        ;FOLD Parameters ;%{h}
        ;Params IlfProvider=kukaroboter.basistech.inlineforms.movement.spline; Kuka.IsGlobalPoint=False; Kuka.PointName=P234; Kuka.BlendingEnabled=False; Kuka.MoveDataName=CPDAT27; Kuka.VelocityPath=0.1; Kuka.VelocityFieldEnabled=True; Kuka.ColDetectFieldEnabled=True; Kuka.CurrentCDSetIndex=0; Kuka.MovementParameterFieldEnabled=True; IlfCommand=SLIN
        ;ENDFOLD
        SLIN XP234 WITH $VEL = SVEL_CP(0.1, , LCPDAT27), $TOOL = STOOL2(FP234), $BASE = SBASE(FP234.BASE_NO), $IPO_MODE = SIPO_MODE(FP234.IPO_FRAME), $LOAD = SLOAD(FP234.TOOL_NO), $ACC = SACC_CP(LCPDAT27), $ORI_TYPE = SORI_TYP(LCPDAT27), $APO = SAPO(LCPDAT27), $JERK = SJERK(LCPDAT27), $COLLMON_TOL_PRO[1] = USE_CM_PRO_VALUES(0)
        ;ENDFOLD
        ;FOLD Gripper SET [1]Gripper1 State=[1]ABIERTA Wait 0.2[s] Check with Strategy 1 ;%{PE}
        ;FOLD Parameters Parameters ;%{h}
        ;Params IlfProvider=GripperTech.GripperSet;setgripper=1;setstate=1;setcont=nocont;waittime=0.2;errorstrategy=1
        ;ENDFOLD
        GRPg_SetStateAndCheck(1, 1, 0.2, 1)
        ;ENDFOLD
        ;FOLD SLIN P134 Vel=0.1 m/s CPDAT28 Tool[1]:SMC Base[0] ;%{PE}
        ;FOLD Parameters ;%{h}
        ;Params IlfProvider=kukaroboter.basistech.inlineforms.movement.spline; Kuka.IsGlobalPoint=False; Kuka.PointName=P134; Kuka.BlendingEnabled=False; Kuka.MoveDataName=CPDAT28; Kuka.VelocityPath=0.1; Kuka.VelocityFieldEnabled=True; Kuka.ColDetectFieldEnabled=True; Kuka.CurrentCDSetIndex=0; Kuka.MovementParameterFieldEnabled=True; IlfCommand=SLIN
        ;ENDFOLD
        SLIN XP134 WITH $VEL = SVEL_CP(0.1, , LCPDAT28), $TOOL = STOOL2(FP134), $BASE = SBASE(FP134.BASE_NO), $IPO_MODE = SIPO_MODE(FP134.IPO_FRAME), $LOAD = SLOAD(FP134.TOOL_NO), $ACC = SACC_CP(LCPDAT28), $ORI_TYPE = SORI_TYP(LCPDAT28), $APO = SAPO(LCPDAT28), $JERK = SJERK(LCPDAT28), $COLLMON_TOL_PRO[1] = USE_CM_PRO_VALUES(0)
        ;ENDFOLD
        ;FOLD SPTP P600 Vel=100 % PDAT1 Tool[1]:SMC Base[0] ;%{PE}
        ;FOLD Parameters ;%{h}
        ;Params IlfProvider=kukaroboter.basistech.inlineforms.movement.spline; Kuka.IsGlobalPoint=False; Kuka.PointName=P600; Kuka.BlendingEnabled=False; Kuka.MoveDataPtpName=PDAT1; Kuka.VelocityPtp=100; Kuka.VelocityFieldEnabled=True; Kuka.ColDetectFieldEnabled=True; Kuka.CurrentCDSetIndex=0; Kuka.MovementParameterFieldEnabled=True; IlfCommand=SPTP
        ;ENDFOLD
        SPTP XP600 WITH $VEL_AXIS[1] = SVEL_JOINT(100.0), $TOOL = STOOL2(FP600), $BASE = SBASE(FP600.BASE_NO), $IPO_MODE = SIPO_MODE(FP600.IPO_FRAME), $LOAD = SLOAD(FP600.TOOL_NO), $ACC_AXIS[1] = SACC_JOINT(PPDAT1), $APO = SAPO_PTP(PPDAT1), $GEAR_JERK[1] = SGEAR_JERK(PPDAT1), $COLLMON_TOL_PRO[1] = USE_CM_PRO_VALUES(0)
        ;ENDFOLD
        ;FOLD SLIN P601 Vel=0.1 m/s CPDAT27 Tool[1]:SMC Base[0] ;%{PE}
        ;FOLD Parameters ;%{h}
        ;Params IlfProvider=kukaroboter.basistech.inlineforms.movement.spline; Kuka.IsGlobalPoint=False; Kuka.PointName=P601; Kuka.BlendingEnabled=False; Kuka.MoveDataName=CPDAT27; Kuka.VelocityPath=0.1; Kuka.VelocityFieldEnabled=True; Kuka.ColDetectFieldEnabled=True; Kuka.CurrentCDSetIndex=0; Kuka.MovementParameterFieldEnabled=True; IlfCommand=SLIN
        ;ENDFOLD
        SLIN XP601 WITH $VEL = SVEL_CP(0.1, , LCPDAT27), $TOOL = STOOL2(FP601), $BASE = SBASE(FP601.BASE_NO), $IPO_MODE = SIPO_MODE(FP601.IPO_FRAME), $LOAD = SLOAD(FP601.TOOL_NO), $ACC = SACC_CP(LCPDAT27), $ORI_TYPE = SORI_TYP(LCPDAT27), $APO = SAPO(LCPDAT27), $JERK = SJERK(LCPDAT27), $COLLMON_TOL_PRO[1] = USE_CM_PRO_VALUES(0)
        ;ENDFOLD
        ;FOLD SLIN P602 Vel=0.1 m/s CPDAT27 Tool[1]:SMC Base[0] ;%{PE}
        ;FOLD Parameters ;%{h}
        ;Params IlfProvider=kukaroboter.basistech.inlineforms.movement.spline; Kuka.IsGlobalPoint=False; Kuka.PointName=P602; Kuka.BlendingEnabled=False; Kuka.MoveDataName=CPDAT27; Kuka.VelocityPath=0.1; Kuka.VelocityFieldEnabled=True; Kuka.ColDetectFieldEnabled=True; Kuka.CurrentCDSetIndex=0; Kuka.MovementParameterFieldEnabled=True; IlfCommand=SLIN
        ;ENDFOLD
        SLIN XP602 WITH $VEL = SVEL_CP(0.1, , LCPDAT27), $TOOL = STOOL2(FP602), $BASE = SBASE(FP602.BASE_NO), $IPO_MODE = SIPO_MODE(FP602.IPO_FRAME), $LOAD = SLOAD(FP602.TOOL_NO), $ACC = SACC_CP(LCPDAT27), $ORI_TYPE = SORI_TYP(LCPDAT27), $APO = SAPO(LCPDAT27), $JERK = SJERK(LCPDAT27), $COLLMON_TOL_PRO[1] = USE_CM_PRO_VALUES(0)
        ;ENDFOLD
      ENDIF

      IF finalPosition == 35 THEN
        ;FOLD SPTP P135 Vel=100 % PDAT1 Tool[1]:SMC Base[0] ;%{PE}
        ;FOLD Parameters ;%{h}
        ;Params IlfProvider=kukaroboter.basistech.inlineforms.movement.spline; Kuka.IsGlobalPoint=False; Kuka.PointName=P135; Kuka.BlendingEnabled=False; Kuka.MoveDataPtpName=PDAT1; Kuka.VelocityPtp=100; Kuka.VelocityFieldEnabled=True; Kuka.ColDetectFieldEnabled=True; Kuka.CurrentCDSetIndex=0; Kuka.MovementParameterFieldEnabled=True; IlfCommand=SPTP
        ;ENDFOLD
        SPTP XP135 WITH $VEL_AXIS[1] = SVEL_JOINT(100.0), $TOOL = STOOL2(FP135), $BASE = SBASE(FP135.BASE_NO), $IPO_MODE = SIPO_MODE(FP135.IPO_FRAME), $LOAD = SLOAD(FP135.TOOL_NO), $ACC_AXIS[1] = SACC_JOINT(PPDAT1), $APO = SAPO_PTP(PPDAT1), $GEAR_JERK[1] = SGEAR_JERK(PPDAT1), $COLLMON_TOL_PRO[1] = USE_CM_PRO_VALUES(0)
        ;ENDFOLD
        ;FOLD SLIN P235 Vel=0.1 m/s CPDAT27 Tool[1]:SMC Base[0] ;%{PE}
        ;FOLD Parameters ;%{h}
        ;Params IlfProvider=kukaroboter.basistech.inlineforms.movement.spline; Kuka.IsGlobalPoint=False; Kuka.PointName=P235; Kuka.BlendingEnabled=False; Kuka.MoveDataName=CPDAT27; Kuka.VelocityPath=0.1; Kuka.VelocityFieldEnabled=True; Kuka.ColDetectFieldEnabled=True; Kuka.CurrentCDSetIndex=0; Kuka.MovementParameterFieldEnabled=True; IlfCommand=SLIN
        ;ENDFOLD
        SLIN XP235 WITH $VEL = SVEL_CP(0.1, , LCPDAT27), $TOOL = STOOL2(FP235), $BASE = SBASE(FP235.BASE_NO), $IPO_MODE = SIPO_MODE(FP235.IPO_FRAME), $LOAD = SLOAD(FP235.TOOL_NO), $ACC = SACC_CP(LCPDAT27), $ORI_TYPE = SORI_TYP(LCPDAT27), $APO = SAPO(LCPDAT27), $JERK = SJERK(LCPDAT27), $COLLMON_TOL_PRO[1] = USE_CM_PRO_VALUES(0)
        ;ENDFOLD
        ;FOLD Gripper SET [1]Gripper1 State=[1]ABIERTA Wait 0.2[s] Check with Strategy 1 ;%{PE}
        ;FOLD Parameters Parameters ;%{h}
        ;Params IlfProvider=GripperTech.GripperSet;setgripper=1;setstate=1;setcont=nocont;waittime=0.2;errorstrategy=1
        ;ENDFOLD
        GRPg_SetStateAndCheck(1, 1, 0.2, 1)
        ;ENDFOLD
        ;FOLD SLIN P135 Vel=0.1 m/s CPDAT28 Tool[1]:SMC Base[0] ;%{PE}
        ;FOLD Parameters ;%{h}
        ;Params IlfProvider=kukaroboter.basistech.inlineforms.movement.spline; Kuka.IsGlobalPoint=False; Kuka.PointName=P135; Kuka.BlendingEnabled=False; Kuka.MoveDataName=CPDAT28; Kuka.VelocityPath=0.1; Kuka.VelocityFieldEnabled=True; Kuka.ColDetectFieldEnabled=True; Kuka.CurrentCDSetIndex=0; Kuka.MovementParameterFieldEnabled=True; IlfCommand=SLIN
        ;ENDFOLD
        SLIN XP135 WITH $VEL = SVEL_CP(0.1, , LCPDAT28), $TOOL = STOOL2(FP135), $BASE = SBASE(FP135.BASE_NO), $IPO_MODE = SIPO_MODE(FP135.IPO_FRAME), $LOAD = SLOAD(FP135.TOOL_NO), $ACC = SACC_CP(LCPDAT28), $ORI_TYPE = SORI_TYP(LCPDAT28), $APO = SAPO(LCPDAT28), $JERK = SJERK(LCPDAT28), $COLLMON_TOL_PRO[1] = USE_CM_PRO_VALUES(0)
        ;ENDFOLD
        ;FOLD SPTP P600 Vel=100 % PDAT1 Tool[1]:SMC Base[0] ;%{PE}
        ;FOLD Parameters ;%{h}
        ;Params IlfProvider=kukaroboter.basistech.inlineforms.movement.spline; Kuka.IsGlobalPoint=False; Kuka.PointName=P600; Kuka.BlendingEnabled=False; Kuka.MoveDataPtpName=PDAT1; Kuka.VelocityPtp=100; Kuka.VelocityFieldEnabled=True; Kuka.ColDetectFieldEnabled=True; Kuka.CurrentCDSetIndex=0; Kuka.MovementParameterFieldEnabled=True; IlfCommand=SPTP
        ;ENDFOLD
        SPTP XP600 WITH $VEL_AXIS[1] = SVEL_JOINT(100.0), $TOOL = STOOL2(FP600), $BASE = SBASE(FP600.BASE_NO), $IPO_MODE = SIPO_MODE(FP600.IPO_FRAME), $LOAD = SLOAD(FP600.TOOL_NO), $ACC_AXIS[1] = SACC_JOINT(PPDAT1), $APO = SAPO_PTP(PPDAT1), $GEAR_JERK[1] = SGEAR_JERK(PPDAT1), $COLLMON_TOL_PRO[1] = USE_CM_PRO_VALUES(0)
        ;ENDFOLD
        ;FOLD SLIN P601 Vel=0.1 m/s CPDAT27 Tool[1]:SMC Base[0] ;%{PE}
        ;FOLD Parameters ;%{h}
        ;Params IlfProvider=kukaroboter.basistech.inlineforms.movement.spline; Kuka.IsGlobalPoint=False; Kuka.PointName=P601; Kuka.BlendingEnabled=False; Kuka.MoveDataName=CPDAT27; Kuka.VelocityPath=0.1; Kuka.VelocityFieldEnabled=True; Kuka.ColDetectFieldEnabled=True; Kuka.CurrentCDSetIndex=0; Kuka.MovementParameterFieldEnabled=True; IlfCommand=SLIN
        ;ENDFOLD
        SLIN XP601 WITH $VEL = SVEL_CP(0.1, , LCPDAT27), $TOOL = STOOL2(FP601), $BASE = SBASE(FP601.BASE_NO), $IPO_MODE = SIPO_MODE(FP601.IPO_FRAME), $LOAD = SLOAD(FP601.TOOL_NO), $ACC = SACC_CP(LCPDAT27), $ORI_TYPE = SORI_TYP(LCPDAT27), $APO = SAPO(LCPDAT27), $JERK = SJERK(LCPDAT27), $COLLMON_TOL_PRO[1] = USE_CM_PRO_VALUES(0)
        ;ENDFOLD
        ;FOLD SLIN P602 Vel=0.1 m/s CPDAT27 Tool[1]:SMC Base[0] ;%{PE}
        ;FOLD Parameters ;%{h}
        ;Params IlfProvider=kukaroboter.basistech.inlineforms.movement.spline; Kuka.IsGlobalPoint=False; Kuka.PointName=P602; Kuka.BlendingEnabled=False; Kuka.MoveDataName=CPDAT27; Kuka.VelocityPath=0.1; Kuka.VelocityFieldEnabled=True; Kuka.ColDetectFieldEnabled=True; Kuka.CurrentCDSetIndex=0; Kuka.MovementParameterFieldEnabled=True; IlfCommand=SLIN
        ;ENDFOLD
        SLIN XP602 WITH $VEL = SVEL_CP(0.1, , LCPDAT27), $TOOL = STOOL2(FP602), $BASE = SBASE(FP602.BASE_NO), $IPO_MODE = SIPO_MODE(FP602.IPO_FRAME), $LOAD = SLOAD(FP602.TOOL_NO), $ACC = SACC_CP(LCPDAT27), $ORI_TYPE = SORI_TYP(LCPDAT27), $APO = SAPO(LCPDAT27), $JERK = SJERK(LCPDAT27), $COLLMON_TOL_PRO[1] = USE_CM_PRO_VALUES(0)
        ;ENDFOLD
      ENDIF

      IF finalPosition == 36 THEN
        ;FOLD SPTP P136 Vel=100 % PDAT1 Tool[1]:SMC Base[0] ;%{PE}
        ;FOLD Parameters ;%{h}
        ;Params IlfProvider=kukaroboter.basistech.inlineforms.movement.spline; Kuka.IsGlobalPoint=False; Kuka.PointName=P136; Kuka.BlendingEnabled=False; Kuka.MoveDataPtpName=PDAT1; Kuka.VelocityPtp=100; Kuka.VelocityFieldEnabled=True; Kuka.ColDetectFieldEnabled=True; Kuka.CurrentCDSetIndex=0; Kuka.MovementParameterFieldEnabled=True; IlfCommand=SPTP
        ;ENDFOLD
        SPTP XP136 WITH $VEL_AXIS[1] = SVEL_JOINT(100.0), $TOOL = STOOL2(FP136), $BASE = SBASE(FP136.BASE_NO), $IPO_MODE = SIPO_MODE(FP136.IPO_FRAME), $LOAD = SLOAD(FP136.TOOL_NO), $ACC_AXIS[1] = SACC_JOINT(PPDAT1), $APO = SAPO_PTP(PPDAT1), $GEAR_JERK[1] = SGEAR_JERK(PPDAT1), $COLLMON_TOL_PRO[1] = USE_CM_PRO_VALUES(0)
        ;ENDFOLD
        ;FOLD SLIN P236 Vel=0.1 m/s CPDAT27 Tool[1]:SMC Base[0] ;%{PE}
        ;FOLD Parameters ;%{h}
        ;Params IlfProvider=kukaroboter.basistech.inlineforms.movement.spline; Kuka.IsGlobalPoint=False; Kuka.PointName=P236; Kuka.BlendingEnabled=False; Kuka.MoveDataName=CPDAT27; Kuka.VelocityPath=0.1; Kuka.VelocityFieldEnabled=True; Kuka.ColDetectFieldEnabled=True; Kuka.CurrentCDSetIndex=0; Kuka.MovementParameterFieldEnabled=True; IlfCommand=SLIN
        ;ENDFOLD
        SLIN XP236 WITH $VEL = SVEL_CP(0.1, , LCPDAT27), $TOOL = STOOL2(FP236), $BASE = SBASE(FP236.BASE_NO), $IPO_MODE = SIPO_MODE(FP236.IPO_FRAME), $LOAD = SLOAD(FP236.TOOL_NO), $ACC = SACC_CP(LCPDAT27), $ORI_TYPE = SORI_TYP(LCPDAT27), $APO = SAPO(LCPDAT27), $JERK = SJERK(LCPDAT27), $COLLMON_TOL_PRO[1] = USE_CM_PRO_VALUES(0)
        ;ENDFOLD
        ;FOLD Gripper SET [1]Gripper1 State=[1]ABIERTA Wait 0.2[s] Check with Strategy 1 ;%{PE}
        ;FOLD Parameters Parameters ;%{h}
        ;Params IlfProvider=GripperTech.GripperSet;setgripper=1;setstate=1;setcont=nocont;waittime=0.2;errorstrategy=1
        ;ENDFOLD
        GRPg_SetStateAndCheck(1, 1, 0.2, 1)
        ;ENDFOLD
        ;FOLD SLIN P136 Vel=0.1 m/s CPDAT28 Tool[1]:SMC Base[0] ;%{PE}
        ;FOLD Parameters ;%{h}
        ;Params IlfProvider=kukaroboter.basistech.inlineforms.movement.spline; Kuka.IsGlobalPoint=False; Kuka.PointName=P136; Kuka.BlendingEnabled=False; Kuka.MoveDataName=CPDAT28; Kuka.VelocityPath=0.1; Kuka.VelocityFieldEnabled=True; Kuka.ColDetectFieldEnabled=True; Kuka.CurrentCDSetIndex=0; Kuka.MovementParameterFieldEnabled=True; IlfCommand=SLIN
        ;ENDFOLD
        SLIN XP136 WITH $VEL = SVEL_CP(0.1, , LCPDAT28), $TOOL = STOOL2(FP136), $BASE = SBASE(FP136.BASE_NO), $IPO_MODE = SIPO_MODE(FP136.IPO_FRAME), $LOAD = SLOAD(FP136.TOOL_NO), $ACC = SACC_CP(LCPDAT28), $ORI_TYPE = SORI_TYP(LCPDAT28), $APO = SAPO(LCPDAT28), $JERK = SJERK(LCPDAT28), $COLLMON_TOL_PRO[1] = USE_CM_PRO_VALUES(0)
        ;ENDFOLD
        ;FOLD SPTP P600 Vel=100 % PDAT1 Tool[1]:SMC Base[0] ;%{PE}
        ;FOLD Parameters ;%{h}
        ;Params IlfProvider=kukaroboter.basistech.inlineforms.movement.spline; Kuka.IsGlobalPoint=False; Kuka.PointName=P600; Kuka.BlendingEnabled=False; Kuka.MoveDataPtpName=PDAT1; Kuka.VelocityPtp=100; Kuka.VelocityFieldEnabled=True; Kuka.ColDetectFieldEnabled=True; Kuka.CurrentCDSetIndex=0; Kuka.MovementParameterFieldEnabled=True; IlfCommand=SPTP
        ;ENDFOLD
        SPTP XP600 WITH $VEL_AXIS[1] = SVEL_JOINT(100.0), $TOOL = STOOL2(FP600), $BASE = SBASE(FP600.BASE_NO), $IPO_MODE = SIPO_MODE(FP600.IPO_FRAME), $LOAD = SLOAD(FP600.TOOL_NO), $ACC_AXIS[1] = SACC_JOINT(PPDAT1), $APO = SAPO_PTP(PPDAT1), $GEAR_JERK[1] = SGEAR_JERK(PPDAT1), $COLLMON_TOL_PRO[1] = USE_CM_PRO_VALUES(0)
        ;ENDFOLD
        ;FOLD SLIN P601 Vel=0.1 m/s CPDAT27 Tool[1]:SMC Base[0] ;%{PE}
        ;FOLD Parameters ;%{h}
        ;Params IlfProvider=kukaroboter.basistech.inlineforms.movement.spline; Kuka.IsGlobalPoint=False; Kuka.PointName=P601; Kuka.BlendingEnabled=False; Kuka.MoveDataName=CPDAT27; Kuka.VelocityPath=0.1; Kuka.VelocityFieldEnabled=True; Kuka.ColDetectFieldEnabled=True; Kuka.CurrentCDSetIndex=0; Kuka.MovementParameterFieldEnabled=True; IlfCommand=SLIN
        ;ENDFOLD
        SLIN XP601 WITH $VEL = SVEL_CP(0.1, , LCPDAT27), $TOOL = STOOL2(FP601), $BASE = SBASE(FP601.BASE_NO), $IPO_MODE = SIPO_MODE(FP601.IPO_FRAME), $LOAD = SLOAD(FP601.TOOL_NO), $ACC = SACC_CP(LCPDAT27), $ORI_TYPE = SORI_TYP(LCPDAT27), $APO = SAPO(LCPDAT27), $JERK = SJERK(LCPDAT27), $COLLMON_TOL_PRO[1] = USE_CM_PRO_VALUES(0)
        ;ENDFOLD
        ;FOLD SLIN P602 Vel=0.1 m/s CPDAT27 Tool[1]:SMC Base[0] ;%{PE}
        ;FOLD Parameters ;%{h}
        ;Params IlfProvider=kukaroboter.basistech.inlineforms.movement.spline; Kuka.IsGlobalPoint=False; Kuka.PointName=P602; Kuka.BlendingEnabled=False; Kuka.MoveDataName=CPDAT27; Kuka.VelocityPath=0.1; Kuka.VelocityFieldEnabled=True; Kuka.ColDetectFieldEnabled=True; Kuka.CurrentCDSetIndex=0; Kuka.MovementParameterFieldEnabled=True; IlfCommand=SLIN
        ;ENDFOLD
        SLIN XP602 WITH $VEL = SVEL_CP(0.1, , LCPDAT27), $TOOL = STOOL2(FP602), $BASE = SBASE(FP602.BASE_NO), $IPO_MODE = SIPO_MODE(FP602.IPO_FRAME), $LOAD = SLOAD(FP602.TOOL_NO), $ACC = SACC_CP(LCPDAT27), $ORI_TYPE = SORI_TYP(LCPDAT27), $APO = SAPO(LCPDAT27), $JERK = SJERK(LCPDAT27), $COLLMON_TOL_PRO[1] = USE_CM_PRO_VALUES(0)
        ;ENDFOLD
      ENDIF

      IF finalPosition == 37 THEN
        ;FOLD SPTP P137 Vel=100 % PDAT1 Tool[1]:SMC Base[0] ;%{PE}
        ;FOLD Parameters ;%{h}
        ;Params IlfProvider=kukaroboter.basistech.inlineforms.movement.spline; Kuka.IsGlobalPoint=False; Kuka.PointName=P137; Kuka.BlendingEnabled=False; Kuka.MoveDataPtpName=PDAT1; Kuka.VelocityPtp=100; Kuka.VelocityFieldEnabled=True; Kuka.ColDetectFieldEnabled=True; Kuka.CurrentCDSetIndex=0; Kuka.MovementParameterFieldEnabled=True; IlfCommand=SPTP
        ;ENDFOLD
        SPTP XP137 WITH $VEL_AXIS[1] = SVEL_JOINT(100.0), $TOOL = STOOL2(FP137), $BASE = SBASE(FP137.BASE_NO), $IPO_MODE = SIPO_MODE(FP137.IPO_FRAME), $LOAD = SLOAD(FP137.TOOL_NO), $ACC_AXIS[1] = SACC_JOINT(PPDAT1), $APO = SAPO_PTP(PPDAT1), $GEAR_JERK[1] = SGEAR_JERK(PPDAT1), $COLLMON_TOL_PRO[1] = USE_CM_PRO_VALUES(0)
        ;ENDFOLD
        ;FOLD SLIN P237 Vel=0.1 m/s CPDAT27 Tool[1]:SMC Base[0] ;%{PE}
        ;FOLD Parameters ;%{h}
        ;Params IlfProvider=kukaroboter.basistech.inlineforms.movement.spline; Kuka.IsGlobalPoint=False; Kuka.PointName=P237; Kuka.BlendingEnabled=False; Kuka.MoveDataName=CPDAT27; Kuka.VelocityPath=0.1; Kuka.VelocityFieldEnabled=True; Kuka.ColDetectFieldEnabled=True; Kuka.CurrentCDSetIndex=0; Kuka.MovementParameterFieldEnabled=True; IlfCommand=SLIN
        ;ENDFOLD
        SLIN XP237 WITH $VEL = SVEL_CP(0.1, , LCPDAT27), $TOOL = STOOL2(FP237), $BASE = SBASE(FP237.BASE_NO), $IPO_MODE = SIPO_MODE(FP237.IPO_FRAME), $LOAD = SLOAD(FP237.TOOL_NO), $ACC = SACC_CP(LCPDAT27), $ORI_TYPE = SORI_TYP(LCPDAT27), $APO = SAPO(LCPDAT27), $JERK = SJERK(LCPDAT27), $COLLMON_TOL_PRO[1] = USE_CM_PRO_VALUES(0)
        ;ENDFOLD
        ;FOLD Gripper SET [1]Gripper1 State=[1]ABIERTA Wait 0.2[s] Check with Strategy 1 ;%{PE}
        ;FOLD Parameters Parameters ;%{h}
        ;Params IlfProvider=GripperTech.GripperSet;setgripper=1;setstate=1;setcont=nocont;waittime=0.2;errorstrategy=1
        ;ENDFOLD
        GRPg_SetStateAndCheck(1, 1, 0.2, 1)
        ;ENDFOLD
        ;FOLD SLIN P137 Vel=0.1 m/s CPDAT28 Tool[1]:SMC Base[0] ;%{PE}
        ;FOLD Parameters ;%{h}
        ;Params IlfProvider=kukaroboter.basistech.inlineforms.movement.spline; Kuka.IsGlobalPoint=False; Kuka.PointName=P137; Kuka.BlendingEnabled=False; Kuka.MoveDataName=CPDAT28; Kuka.VelocityPath=0.1; Kuka.VelocityFieldEnabled=True; Kuka.ColDetectFieldEnabled=True; Kuka.CurrentCDSetIndex=0; Kuka.MovementParameterFieldEnabled=True; IlfCommand=SLIN
        ;ENDFOLD
        SLIN XP137 WITH $VEL = SVEL_CP(0.1, , LCPDAT28), $TOOL = STOOL2(FP137), $BASE = SBASE(FP137.BASE_NO), $IPO_MODE = SIPO_MODE(FP137.IPO_FRAME), $LOAD = SLOAD(FP137.TOOL_NO), $ACC = SACC_CP(LCPDAT28), $ORI_TYPE = SORI_TYP(LCPDAT28), $APO = SAPO(LCPDAT28), $JERK = SJERK(LCPDAT28), $COLLMON_TOL_PRO[1] = USE_CM_PRO_VALUES(0)
        ;ENDFOLD
        ;FOLD SPTP P600 Vel=100 % PDAT1 Tool[1]:SMC Base[0] ;%{PE}
        ;FOLD Parameters ;%{h}
        ;Params IlfProvider=kukaroboter.basistech.inlineforms.movement.spline; Kuka.IsGlobalPoint=False; Kuka.PointName=P600; Kuka.BlendingEnabled=False; Kuka.MoveDataPtpName=PDAT1; Kuka.VelocityPtp=100; Kuka.VelocityFieldEnabled=True; Kuka.ColDetectFieldEnabled=True; Kuka.CurrentCDSetIndex=0; Kuka.MovementParameterFieldEnabled=True; IlfCommand=SPTP
        ;ENDFOLD
        SPTP XP600 WITH $VEL_AXIS[1] = SVEL_JOINT(100.0), $TOOL = STOOL2(FP600), $BASE = SBASE(FP600.BASE_NO), $IPO_MODE = SIPO_MODE(FP600.IPO_FRAME), $LOAD = SLOAD(FP600.TOOL_NO), $ACC_AXIS[1] = SACC_JOINT(PPDAT1), $APO = SAPO_PTP(PPDAT1), $GEAR_JERK[1] = SGEAR_JERK(PPDAT1), $COLLMON_TOL_PRO[1] = USE_CM_PRO_VALUES(0)
        ;ENDFOLD
        ;FOLD SLIN P601 Vel=0.1 m/s CPDAT27 Tool[1]:SMC Base[0] ;%{PE}
        ;FOLD Parameters ;%{h}
        ;Params IlfProvider=kukaroboter.basistech.inlineforms.movement.spline; Kuka.IsGlobalPoint=False; Kuka.PointName=P601; Kuka.BlendingEnabled=False; Kuka.MoveDataName=CPDAT27; Kuka.VelocityPath=0.1; Kuka.VelocityFieldEnabled=True; Kuka.ColDetectFieldEnabled=True; Kuka.CurrentCDSetIndex=0; Kuka.MovementParameterFieldEnabled=True; IlfCommand=SLIN
        ;ENDFOLD
        SLIN XP601 WITH $VEL = SVEL_CP(0.1, , LCPDAT27), $TOOL = STOOL2(FP601), $BASE = SBASE(FP601.BASE_NO), $IPO_MODE = SIPO_MODE(FP601.IPO_FRAME), $LOAD = SLOAD(FP601.TOOL_NO), $ACC = SACC_CP(LCPDAT27), $ORI_TYPE = SORI_TYP(LCPDAT27), $APO = SAPO(LCPDAT27), $JERK = SJERK(LCPDAT27), $COLLMON_TOL_PRO[1] = USE_CM_PRO_VALUES(0)
        ;ENDFOLD
        ;FOLD SLIN P602 Vel=0.1 m/s CPDAT27 Tool[1]:SMC Base[0] ;%{PE}
        ;FOLD Parameters ;%{h}
        ;Params IlfProvider=kukaroboter.basistech.inlineforms.movement.spline; Kuka.IsGlobalPoint=False; Kuka.PointName=P602; Kuka.BlendingEnabled=False; Kuka.MoveDataName=CPDAT27; Kuka.VelocityPath=0.1; Kuka.VelocityFieldEnabled=True; Kuka.ColDetectFieldEnabled=True; Kuka.CurrentCDSetIndex=0; Kuka.MovementParameterFieldEnabled=True; IlfCommand=SLIN
        ;ENDFOLD
        SLIN XP602 WITH $VEL = SVEL_CP(0.1, , LCPDAT27), $TOOL = STOOL2(FP602), $BASE = SBASE(FP602.BASE_NO), $IPO_MODE = SIPO_MODE(FP602.IPO_FRAME), $LOAD = SLOAD(FP602.TOOL_NO), $ACC = SACC_CP(LCPDAT27), $ORI_TYPE = SORI_TYP(LCPDAT27), $APO = SAPO(LCPDAT27), $JERK = SJERK(LCPDAT27), $COLLMON_TOL_PRO[1] = USE_CM_PRO_VALUES(0)
        ;ENDFOLD
      ENDIF

      IF finalPosition == 38 THEN
        ;FOLD SPTP P138 Vel=100 % PDAT1 Tool[1]:SMC Base[0] ;%{PE}
        ;FOLD Parameters ;%{h}
        ;Params IlfProvider=kukaroboter.basistech.inlineforms.movement.spline; Kuka.IsGlobalPoint=False; Kuka.PointName=P138; Kuka.BlendingEnabled=False; Kuka.MoveDataPtpName=PDAT1; Kuka.VelocityPtp=100; Kuka.VelocityFieldEnabled=True; Kuka.ColDetectFieldEnabled=True; Kuka.CurrentCDSetIndex=0; Kuka.MovementParameterFieldEnabled=True; IlfCommand=SPTP
        ;ENDFOLD
        SPTP XP138 WITH $VEL_AXIS[1] = SVEL_JOINT(100.0), $TOOL = STOOL2(FP138), $BASE = SBASE(FP138.BASE_NO), $IPO_MODE = SIPO_MODE(FP138.IPO_FRAME), $LOAD = SLOAD(FP138.TOOL_NO), $ACC_AXIS[1] = SACC_JOINT(PPDAT1), $APO = SAPO_PTP(PPDAT1), $GEAR_JERK[1] = SGEAR_JERK(PPDAT1), $COLLMON_TOL_PRO[1] = USE_CM_PRO_VALUES(0)
        ;ENDFOLD
        ;FOLD SLIN P238 Vel=0.1 m/s CPDAT27 Tool[1]:SMC Base[0] ;%{PE}
        ;FOLD Parameters ;%{h}
        ;Params IlfProvider=kukaroboter.basistech.inlineforms.movement.spline; Kuka.IsGlobalPoint=False; Kuka.PointName=P238; Kuka.BlendingEnabled=False; Kuka.MoveDataName=CPDAT27; Kuka.VelocityPath=0.1; Kuka.VelocityFieldEnabled=True; Kuka.ColDetectFieldEnabled=True; Kuka.CurrentCDSetIndex=0; Kuka.MovementParameterFieldEnabled=True; IlfCommand=SLIN
        ;ENDFOLD
        SLIN XP238 WITH $VEL = SVEL_CP(0.1, , LCPDAT27), $TOOL = STOOL2(FP238), $BASE = SBASE(FP238.BASE_NO), $IPO_MODE = SIPO_MODE(FP238.IPO_FRAME), $LOAD = SLOAD(FP238.TOOL_NO), $ACC = SACC_CP(LCPDAT27), $ORI_TYPE = SORI_TYP(LCPDAT27), $APO = SAPO(LCPDAT27), $JERK = SJERK(LCPDAT27), $COLLMON_TOL_PRO[1] = USE_CM_PRO_VALUES(0)
        ;ENDFOLD
        ;FOLD Gripper SET [1]Gripper1 State=[1]ABIERTA Wait 0.2[s] Check with Strategy 1 ;%{PE}
        ;FOLD Parameters Parameters ;%{h}
        ;Params IlfProvider=GripperTech.GripperSet;setgripper=1;setstate=1;setcont=nocont;waittime=0.2;errorstrategy=1
        ;ENDFOLD
        GRPg_SetStateAndCheck(1, 1, 0.2, 1)
        ;ENDFOLD
        ;FOLD SLIN P138 Vel=0.1 m/s CPDAT28 Tool[1]:SMC Base[0] ;%{PE}
        ;FOLD Parameters ;%{h}
        ;Params IlfProvider=kukaroboter.basistech.inlineforms.movement.spline; Kuka.IsGlobalPoint=False; Kuka.PointName=P138; Kuka.BlendingEnabled=False; Kuka.MoveDataName=CPDAT28; Kuka.VelocityPath=0.1; Kuka.VelocityFieldEnabled=True; Kuka.ColDetectFieldEnabled=True; Kuka.CurrentCDSetIndex=0; Kuka.MovementParameterFieldEnabled=True; IlfCommand=SLIN
        ;ENDFOLD
        SLIN XP138 WITH $VEL = SVEL_CP(0.1, , LCPDAT28), $TOOL = STOOL2(FP138), $BASE = SBASE(FP138.BASE_NO), $IPO_MODE = SIPO_MODE(FP138.IPO_FRAME), $LOAD = SLOAD(FP138.TOOL_NO), $ACC = SACC_CP(LCPDAT28), $ORI_TYPE = SORI_TYP(LCPDAT28), $APO = SAPO(LCPDAT28), $JERK = SJERK(LCPDAT28), $COLLMON_TOL_PRO[1] = USE_CM_PRO_VALUES(0)
        ;ENDFOLD
        ;FOLD SPTP P600 Vel=100 % PDAT1 Tool[1]:SMC Base[0] ;%{PE}
        ;FOLD Parameters ;%{h}
        ;Params IlfProvider=kukaroboter.basistech.inlineforms.movement.spline; Kuka.IsGlobalPoint=False; Kuka.PointName=P600; Kuka.BlendingEnabled=False; Kuka.MoveDataPtpName=PDAT1; Kuka.VelocityPtp=100; Kuka.VelocityFieldEnabled=True; Kuka.ColDetectFieldEnabled=True; Kuka.CurrentCDSetIndex=0; Kuka.MovementParameterFieldEnabled=True; IlfCommand=SPTP
        ;ENDFOLD
        SPTP XP600 WITH $VEL_AXIS[1] = SVEL_JOINT(100.0), $TOOL = STOOL2(FP600), $BASE = SBASE(FP600.BASE_NO), $IPO_MODE = SIPO_MODE(FP600.IPO_FRAME), $LOAD = SLOAD(FP600.TOOL_NO), $ACC_AXIS[1] = SACC_JOINT(PPDAT1), $APO = SAPO_PTP(PPDAT1), $GEAR_JERK[1] = SGEAR_JERK(PPDAT1), $COLLMON_TOL_PRO[1] = USE_CM_PRO_VALUES(0)
        ;ENDFOLD
        ;FOLD SLIN P601 Vel=0.1 m/s CPDAT27 Tool[1]:SMC Base[0] ;%{PE}
        ;FOLD Parameters ;%{h}
        ;Params IlfProvider=kukaroboter.basistech.inlineforms.movement.spline; Kuka.IsGlobalPoint=False; Kuka.PointName=P601; Kuka.BlendingEnabled=False; Kuka.MoveDataName=CPDAT27; Kuka.VelocityPath=0.1; Kuka.VelocityFieldEnabled=True; Kuka.ColDetectFieldEnabled=True; Kuka.CurrentCDSetIndex=0; Kuka.MovementParameterFieldEnabled=True; IlfCommand=SLIN
        ;ENDFOLD
        SLIN XP601 WITH $VEL = SVEL_CP(0.1, , LCPDAT27), $TOOL = STOOL2(FP601), $BASE = SBASE(FP601.BASE_NO), $IPO_MODE = SIPO_MODE(FP601.IPO_FRAME), $LOAD = SLOAD(FP601.TOOL_NO), $ACC = SACC_CP(LCPDAT27), $ORI_TYPE = SORI_TYP(LCPDAT27), $APO = SAPO(LCPDAT27), $JERK = SJERK(LCPDAT27), $COLLMON_TOL_PRO[1] = USE_CM_PRO_VALUES(0)
        ;ENDFOLD
        ;FOLD SLIN P602 Vel=0.1 m/s CPDAT27 Tool[1]:SMC Base[0] ;%{PE}
        ;FOLD Parameters ;%{h}
        ;Params IlfProvider=kukaroboter.basistech.inlineforms.movement.spline; Kuka.IsGlobalPoint=False; Kuka.PointName=P602; Kuka.BlendingEnabled=False; Kuka.MoveDataName=CPDAT27; Kuka.VelocityPath=0.1; Kuka.VelocityFieldEnabled=True; Kuka.ColDetectFieldEnabled=True; Kuka.CurrentCDSetIndex=0; Kuka.MovementParameterFieldEnabled=True; IlfCommand=SLIN
        ;ENDFOLD
        SLIN XP602 WITH $VEL = SVEL_CP(0.1, , LCPDAT27), $TOOL = STOOL2(FP602), $BASE = SBASE(FP602.BASE_NO), $IPO_MODE = SIPO_MODE(FP602.IPO_FRAME), $LOAD = SLOAD(FP602.TOOL_NO), $ACC = SACC_CP(LCPDAT27), $ORI_TYPE = SORI_TYP(LCPDAT27), $APO = SAPO(LCPDAT27), $JERK = SJERK(LCPDAT27), $COLLMON_TOL_PRO[1] = USE_CM_PRO_VALUES(0)
        ;ENDFOLD
      ENDIF

      IF finalPosition == 39 THEN
        ;FOLD SPTP P139 Vel=100 % PDAT1 Tool[1]:SMC Base[0] ;%{PE}
        ;FOLD Parameters ;%{h}
        ;Params IlfProvider=kukaroboter.basistech.inlineforms.movement.spline; Kuka.IsGlobalPoint=False; Kuka.PointName=P139; Kuka.BlendingEnabled=False; Kuka.MoveDataPtpName=PDAT1; Kuka.VelocityPtp=100; Kuka.VelocityFieldEnabled=True; Kuka.ColDetectFieldEnabled=True; Kuka.CurrentCDSetIndex=0; Kuka.MovementParameterFieldEnabled=True; IlfCommand=SPTP
        ;ENDFOLD
        SPTP XP139 WITH $VEL_AXIS[1] = SVEL_JOINT(100.0), $TOOL = STOOL2(FP139), $BASE = SBASE(FP139.BASE_NO), $IPO_MODE = SIPO_MODE(FP139.IPO_FRAME), $LOAD = SLOAD(FP139.TOOL_NO), $ACC_AXIS[1] = SACC_JOINT(PPDAT1), $APO = SAPO_PTP(PPDAT1), $GEAR_JERK[1] = SGEAR_JERK(PPDAT1), $COLLMON_TOL_PRO[1] = USE_CM_PRO_VALUES(0)
        ;ENDFOLD
        ;FOLD SLIN P239 Vel=0.1 m/s CPDAT27 Tool[1]:SMC Base[0] ;%{PE}
        ;FOLD Parameters ;%{h}
        ;Params IlfProvider=kukaroboter.basistech.inlineforms.movement.spline; Kuka.IsGlobalPoint=False; Kuka.PointName=P239; Kuka.BlendingEnabled=False; Kuka.MoveDataName=CPDAT27; Kuka.VelocityPath=0.1; Kuka.VelocityFieldEnabled=True; Kuka.ColDetectFieldEnabled=True; Kuka.CurrentCDSetIndex=0; Kuka.MovementParameterFieldEnabled=True; IlfCommand=SLIN
        ;ENDFOLD
        SLIN XP239 WITH $VEL = SVEL_CP(0.1, , LCPDAT27), $TOOL = STOOL2(FP239), $BASE = SBASE(FP239.BASE_NO), $IPO_MODE = SIPO_MODE(FP239.IPO_FRAME), $LOAD = SLOAD(FP239.TOOL_NO), $ACC = SACC_CP(LCPDAT27), $ORI_TYPE = SORI_TYP(LCPDAT27), $APO = SAPO(LCPDAT27), $JERK = SJERK(LCPDAT27), $COLLMON_TOL_PRO[1] = USE_CM_PRO_VALUES(0)
        ;ENDFOLD
        ;FOLD Gripper SET [1]Gripper1 State=[1]ABIERTA Wait 0.2[s] Check with Strategy 1 ;%{PE}
        ;FOLD Parameters Parameters ;%{h}
        ;Params IlfProvider=GripperTech.GripperSet;setgripper=1;setstate=1;setcont=nocont;waittime=0.2;errorstrategy=1
        ;ENDFOLD
        GRPg_SetStateAndCheck(1, 1, 0.2, 1)
        ;ENDFOLD
        ;FOLD SLIN P139 Vel=0.1 m/s CPDAT28 Tool[1]:SMC Base[0] ;%{PE}
        ;FOLD Parameters ;%{h}
        ;Params IlfProvider=kukaroboter.basistech.inlineforms.movement.spline; Kuka.IsGlobalPoint=False; Kuka.PointName=P139; Kuka.BlendingEnabled=False; Kuka.MoveDataName=CPDAT28; Kuka.VelocityPath=0.1; Kuka.VelocityFieldEnabled=True; Kuka.ColDetectFieldEnabled=True; Kuka.CurrentCDSetIndex=0; Kuka.MovementParameterFieldEnabled=True; IlfCommand=SLIN
        ;ENDFOLD
        SLIN XP139 WITH $VEL = SVEL_CP(0.1, , LCPDAT28), $TOOL = STOOL2(FP139), $BASE = SBASE(FP139.BASE_NO), $IPO_MODE = SIPO_MODE(FP139.IPO_FRAME), $LOAD = SLOAD(FP139.TOOL_NO), $ACC = SACC_CP(LCPDAT28), $ORI_TYPE = SORI_TYP(LCPDAT28), $APO = SAPO(LCPDAT28), $JERK = SJERK(LCPDAT28), $COLLMON_TOL_PRO[1] = USE_CM_PRO_VALUES(0)
        ;ENDFOLD
        ;FOLD SPTP P600 Vel=100 % PDAT1 Tool[1]:SMC Base[0] ;%{PE}
        ;FOLD Parameters ;%{h}
        ;Params IlfProvider=kukaroboter.basistech.inlineforms.movement.spline; Kuka.IsGlobalPoint=False; Kuka.PointName=P600; Kuka.BlendingEnabled=False; Kuka.MoveDataPtpName=PDAT1; Kuka.VelocityPtp=100; Kuka.VelocityFieldEnabled=True; Kuka.ColDetectFieldEnabled=True; Kuka.CurrentCDSetIndex=0; Kuka.MovementParameterFieldEnabled=True; IlfCommand=SPTP
        ;ENDFOLD
        SPTP XP600 WITH $VEL_AXIS[1] = SVEL_JOINT(100.0), $TOOL = STOOL2(FP600), $BASE = SBASE(FP600.BASE_NO), $IPO_MODE = SIPO_MODE(FP600.IPO_FRAME), $LOAD = SLOAD(FP600.TOOL_NO), $ACC_AXIS[1] = SACC_JOINT(PPDAT1), $APO = SAPO_PTP(PPDAT1), $GEAR_JERK[1] = SGEAR_JERK(PPDAT1), $COLLMON_TOL_PRO[1] = USE_CM_PRO_VALUES(0)
        ;ENDFOLD
        ;FOLD SLIN P601 Vel=0.1 m/s CPDAT27 Tool[1]:SMC Base[0] ;%{PE}
        ;FOLD Parameters ;%{h}
        ;Params IlfProvider=kukaroboter.basistech.inlineforms.movement.spline; Kuka.IsGlobalPoint=False; Kuka.PointName=P601; Kuka.BlendingEnabled=False; Kuka.MoveDataName=CPDAT27; Kuka.VelocityPath=0.1; Kuka.VelocityFieldEnabled=True; Kuka.ColDetectFieldEnabled=True; Kuka.CurrentCDSetIndex=0; Kuka.MovementParameterFieldEnabled=True; IlfCommand=SLIN
        ;ENDFOLD
        SLIN XP601 WITH $VEL = SVEL_CP(0.1, , LCPDAT27), $TOOL = STOOL2(FP601), $BASE = SBASE(FP601.BASE_NO), $IPO_MODE = SIPO_MODE(FP601.IPO_FRAME), $LOAD = SLOAD(FP601.TOOL_NO), $ACC = SACC_CP(LCPDAT27), $ORI_TYPE = SORI_TYP(LCPDAT27), $APO = SAPO(LCPDAT27), $JERK = SJERK(LCPDAT27), $COLLMON_TOL_PRO[1] = USE_CM_PRO_VALUES(0)
        ;ENDFOLD
        ;FOLD SLIN P602 Vel=0.1 m/s CPDAT27 Tool[1]:SMC Base[0] ;%{PE}
        ;FOLD Parameters ;%{h}
        ;Params IlfProvider=kukaroboter.basistech.inlineforms.movement.spline; Kuka.IsGlobalPoint=False; Kuka.PointName=P602; Kuka.BlendingEnabled=False; Kuka.MoveDataName=CPDAT27; Kuka.VelocityPath=0.1; Kuka.VelocityFieldEnabled=True; Kuka.ColDetectFieldEnabled=True; Kuka.CurrentCDSetIndex=0; Kuka.MovementParameterFieldEnabled=True; IlfCommand=SLIN
        ;ENDFOLD
        SLIN XP602 WITH $VEL = SVEL_CP(0.1, , LCPDAT27), $TOOL = STOOL2(FP602), $BASE = SBASE(FP602.BASE_NO), $IPO_MODE = SIPO_MODE(FP602.IPO_FRAME), $LOAD = SLOAD(FP602.TOOL_NO), $ACC = SACC_CP(LCPDAT27), $ORI_TYPE = SORI_TYP(LCPDAT27), $APO = SAPO(LCPDAT27), $JERK = SJERK(LCPDAT27), $COLLMON_TOL_PRO[1] = USE_CM_PRO_VALUES(0)
        ;ENDFOLD
      ENDIF

      IF finalPosition == 40 THEN
        ;FOLD SPTP P140 Vel=100 % PDAT1 Tool[1]:SMC Base[0] ;%{PE}
        ;FOLD Parameters ;%{h}
        ;Params IlfProvider=kukaroboter.basistech.inlineforms.movement.spline; Kuka.IsGlobalPoint=False; Kuka.PointName=P140; Kuka.BlendingEnabled=False; Kuka.MoveDataPtpName=PDAT1; Kuka.VelocityPtp=100; Kuka.VelocityFieldEnabled=True; Kuka.ColDetectFieldEnabled=True; Kuka.CurrentCDSetIndex=0; Kuka.MovementParameterFieldEnabled=True; IlfCommand=SPTP
        ;ENDFOLD
        SPTP XP140 WITH $VEL_AXIS[1] = SVEL_JOINT(100.0), $TOOL = STOOL2(FP140), $BASE = SBASE(FP140.BASE_NO), $IPO_MODE = SIPO_MODE(FP140.IPO_FRAME), $LOAD = SLOAD(FP140.TOOL_NO), $ACC_AXIS[1] = SACC_JOINT(PPDAT1), $APO = SAPO_PTP(PPDAT1), $GEAR_JERK[1] = SGEAR_JERK(PPDAT1), $COLLMON_TOL_PRO[1] = USE_CM_PRO_VALUES(0)
        ;ENDFOLD
        ;FOLD SLIN P240 Vel=0.1 m/s CPDAT27 Tool[1]:SMC Base[0] ;%{PE}
        ;FOLD Parameters ;%{h}
        ;Params IlfProvider=kukaroboter.basistech.inlineforms.movement.spline; Kuka.IsGlobalPoint=False; Kuka.PointName=P240; Kuka.BlendingEnabled=False; Kuka.MoveDataName=CPDAT27; Kuka.VelocityPath=0.1; Kuka.VelocityFieldEnabled=True; Kuka.ColDetectFieldEnabled=True; Kuka.CurrentCDSetIndex=0; Kuka.MovementParameterFieldEnabled=True; IlfCommand=SLIN
        ;ENDFOLD
        SLIN XP240 WITH $VEL = SVEL_CP(0.1, , LCPDAT27), $TOOL = STOOL2(FP240), $BASE = SBASE(FP240.BASE_NO), $IPO_MODE = SIPO_MODE(FP240.IPO_FRAME), $LOAD = SLOAD(FP240.TOOL_NO), $ACC = SACC_CP(LCPDAT27), $ORI_TYPE = SORI_TYP(LCPDAT27), $APO = SAPO(LCPDAT27), $JERK = SJERK(LCPDAT27), $COLLMON_TOL_PRO[1] = USE_CM_PRO_VALUES(0)
        ;ENDFOLD
        ;FOLD Gripper SET [1]Gripper1 State=[1]ABIERTA Wait 0.2[s] Check with Strategy 1 ;%{PE}
        ;FOLD Parameters Parameters ;%{h}
        ;Params IlfProvider=GripperTech.GripperSet;setgripper=1;setstate=1;setcont=nocont;waittime=0.2;errorstrategy=1
        ;ENDFOLD
        GRPg_SetStateAndCheck(1, 1, 0.2, 1)
        ;ENDFOLD
        ;FOLD SLIN P140 Vel=0.1 m/s CPDAT28 Tool[1]:SMC Base[0] ;%{PE}
        ;FOLD Parameters ;%{h}
        ;Params IlfProvider=kukaroboter.basistech.inlineforms.movement.spline; Kuka.IsGlobalPoint=False; Kuka.PointName=P140; Kuka.BlendingEnabled=False; Kuka.MoveDataName=CPDAT28; Kuka.VelocityPath=0.1; Kuka.VelocityFieldEnabled=True; Kuka.ColDetectFieldEnabled=True; Kuka.CurrentCDSetIndex=0; Kuka.MovementParameterFieldEnabled=True; IlfCommand=SLIN
        ;ENDFOLD
        SLIN XP140 WITH $VEL = SVEL_CP(0.1, , LCPDAT28), $TOOL = STOOL2(FP140), $BASE = SBASE(FP140.BASE_NO), $IPO_MODE = SIPO_MODE(FP140.IPO_FRAME), $LOAD = SLOAD(FP140.TOOL_NO), $ACC = SACC_CP(LCPDAT28), $ORI_TYPE = SORI_TYP(LCPDAT28), $APO = SAPO(LCPDAT28), $JERK = SJERK(LCPDAT28), $COLLMON_TOL_PRO[1] = USE_CM_PRO_VALUES(0)
        ;ENDFOLD
        ;FOLD SPTP P600 Vel=100 % PDAT1 Tool[1]:SMC Base[0] ;%{PE}
        ;FOLD Parameters ;%{h}
        ;Params IlfProvider=kukaroboter.basistech.inlineforms.movement.spline; Kuka.IsGlobalPoint=False; Kuka.PointName=P600; Kuka.BlendingEnabled=False; Kuka.MoveDataPtpName=PDAT1; Kuka.VelocityPtp=100; Kuka.VelocityFieldEnabled=True; Kuka.ColDetectFieldEnabled=True; Kuka.CurrentCDSetIndex=0; Kuka.MovementParameterFieldEnabled=True; IlfCommand=SPTP
        ;ENDFOLD
        SPTP XP600 WITH $VEL_AXIS[1] = SVEL_JOINT(100.0), $TOOL = STOOL2(FP600), $BASE = SBASE(FP600.BASE_NO), $IPO_MODE = SIPO_MODE(FP600.IPO_FRAME), $LOAD = SLOAD(FP600.TOOL_NO), $ACC_AXIS[1] = SACC_JOINT(PPDAT1), $APO = SAPO_PTP(PPDAT1), $GEAR_JERK[1] = SGEAR_JERK(PPDAT1), $COLLMON_TOL_PRO[1] = USE_CM_PRO_VALUES(0)
        ;ENDFOLD
        ;FOLD SLIN P601 Vel=0.1 m/s CPDAT27 Tool[1]:SMC Base[0] ;%{PE}
        ;FOLD Parameters ;%{h}
        ;Params IlfProvider=kukaroboter.basistech.inlineforms.movement.spline; Kuka.IsGlobalPoint=False; Kuka.PointName=P601; Kuka.BlendingEnabled=False; Kuka.MoveDataName=CPDAT27; Kuka.VelocityPath=0.1; Kuka.VelocityFieldEnabled=True; Kuka.ColDetectFieldEnabled=True; Kuka.CurrentCDSetIndex=0; Kuka.MovementParameterFieldEnabled=True; IlfCommand=SLIN
        ;ENDFOLD
        SLIN XP601 WITH $VEL = SVEL_CP(0.1, , LCPDAT27), $TOOL = STOOL2(FP601), $BASE = SBASE(FP601.BASE_NO), $IPO_MODE = SIPO_MODE(FP601.IPO_FRAME), $LOAD = SLOAD(FP601.TOOL_NO), $ACC = SACC_CP(LCPDAT27), $ORI_TYPE = SORI_TYP(LCPDAT27), $APO = SAPO(LCPDAT27), $JERK = SJERK(LCPDAT27), $COLLMON_TOL_PRO[1] = USE_CM_PRO_VALUES(0)
        ;ENDFOLD
        ;FOLD SLIN P602 Vel=0.1 m/s CPDAT27 Tool[1]:SMC Base[0] ;%{PE}
        ;FOLD Parameters ;%{h}
        ;Params IlfProvider=kukaroboter.basistech.inlineforms.movement.spline; Kuka.IsGlobalPoint=False; Kuka.PointName=P602; Kuka.BlendingEnabled=False; Kuka.MoveDataName=CPDAT27; Kuka.VelocityPath=0.1; Kuka.VelocityFieldEnabled=True; Kuka.ColDetectFieldEnabled=True; Kuka.CurrentCDSetIndex=0; Kuka.MovementParameterFieldEnabled=True; IlfCommand=SLIN
        ;ENDFOLD
        SLIN XP602 WITH $VEL = SVEL_CP(0.1, , LCPDAT27), $TOOL = STOOL2(FP602), $BASE = SBASE(FP602.BASE_NO), $IPO_MODE = SIPO_MODE(FP602.IPO_FRAME), $LOAD = SLOAD(FP602.TOOL_NO), $ACC = SACC_CP(LCPDAT27), $ORI_TYPE = SORI_TYP(LCPDAT27), $APO = SAPO(LCPDAT27), $JERK = SJERK(LCPDAT27), $COLLMON_TOL_PRO[1] = USE_CM_PRO_VALUES(0)
        ;ENDFOLD
      ENDIF

      IF finalPosition == 41 THEN
        ;FOLD SPTP P141 Vel=100 % PDAT1 Tool[1]:SMC Base[0] ;%{PE}
        ;FOLD Parameters ;%{h}
        ;Params IlfProvider=kukaroboter.basistech.inlineforms.movement.spline; Kuka.IsGlobalPoint=False; Kuka.PointName=P141; Kuka.BlendingEnabled=False; Kuka.MoveDataPtpName=PDAT1; Kuka.VelocityPtp=100; Kuka.VelocityFieldEnabled=True; Kuka.ColDetectFieldEnabled=True; Kuka.CurrentCDSetIndex=0; Kuka.MovementParameterFieldEnabled=True; IlfCommand=SPTP
        ;ENDFOLD
        SPTP XP141 WITH $VEL_AXIS[1] = SVEL_JOINT(100.0), $TOOL = STOOL2(FP141), $BASE = SBASE(FP141.BASE_NO), $IPO_MODE = SIPO_MODE(FP141.IPO_FRAME), $LOAD = SLOAD(FP141.TOOL_NO), $ACC_AXIS[1] = SACC_JOINT(PPDAT1), $APO = SAPO_PTP(PPDAT1), $GEAR_JERK[1] = SGEAR_JERK(PPDAT1), $COLLMON_TOL_PRO[1] = USE_CM_PRO_VALUES(0)
        ;ENDFOLD
        ;FOLD SLIN P241 Vel=0.1 m/s CPDAT27 Tool[1]:SMC Base[0] ;%{PE}
        ;FOLD Parameters ;%{h}
        ;Params IlfProvider=kukaroboter.basistech.inlineforms.movement.spline; Kuka.IsGlobalPoint=False; Kuka.PointName=P241; Kuka.BlendingEnabled=False; Kuka.MoveDataName=CPDAT27; Kuka.VelocityPath=0.1; Kuka.VelocityFieldEnabled=True; Kuka.ColDetectFieldEnabled=True; Kuka.CurrentCDSetIndex=0; Kuka.MovementParameterFieldEnabled=True; IlfCommand=SLIN
        ;ENDFOLD
        SLIN XP241 WITH $VEL = SVEL_CP(0.1, , LCPDAT27), $TOOL = STOOL2(FP241), $BASE = SBASE(FP241.BASE_NO), $IPO_MODE = SIPO_MODE(FP241.IPO_FRAME), $LOAD = SLOAD(FP241.TOOL_NO), $ACC = SACC_CP(LCPDAT27), $ORI_TYPE = SORI_TYP(LCPDAT27), $APO = SAPO(LCPDAT27), $JERK = SJERK(LCPDAT27), $COLLMON_TOL_PRO[1] = USE_CM_PRO_VALUES(0)
        ;ENDFOLD
        ;FOLD Gripper SET [1]Gripper1 State=[1]ABIERTA Wait 0.2[s] Check with Strategy 1 ;%{PE}
        ;FOLD Parameters Parameters ;%{h}
        ;Params IlfProvider=GripperTech.GripperSet;setgripper=1;setstate=1;setcont=nocont;waittime=0.2;errorstrategy=1
        ;ENDFOLD
        GRPg_SetStateAndCheck(1, 1, 0.2, 1)
        ;ENDFOLD
        ;FOLD SLIN P141 Vel=0.1 m/s CPDAT28 Tool[1]:SMC Base[0] ;%{PE}
        ;FOLD Parameters ;%{h}
        ;Params IlfProvider=kukaroboter.basistech.inlineforms.movement.spline; Kuka.IsGlobalPoint=False; Kuka.PointName=P141; Kuka.BlendingEnabled=False; Kuka.MoveDataName=CPDAT28; Kuka.VelocityPath=0.1; Kuka.VelocityFieldEnabled=True; Kuka.ColDetectFieldEnabled=True; Kuka.CurrentCDSetIndex=0; Kuka.MovementParameterFieldEnabled=True; IlfCommand=SLIN
        ;ENDFOLD
        SLIN XP141 WITH $VEL = SVEL_CP(0.1, , LCPDAT28), $TOOL = STOOL2(FP141), $BASE = SBASE(FP141.BASE_NO), $IPO_MODE = SIPO_MODE(FP141.IPO_FRAME), $LOAD = SLOAD(FP141.TOOL_NO), $ACC = SACC_CP(LCPDAT28), $ORI_TYPE = SORI_TYP(LCPDAT28), $APO = SAPO(LCPDAT28), $JERK = SJERK(LCPDAT28), $COLLMON_TOL_PRO[1] = USE_CM_PRO_VALUES(0)
        ;ENDFOLD
        ;FOLD SPTP P600 Vel=100 % PDAT1 Tool[1]:SMC Base[0] ;%{PE}
        ;FOLD Parameters ;%{h}
        ;Params IlfProvider=kukaroboter.basistech.inlineforms.movement.spline; Kuka.IsGlobalPoint=False; Kuka.PointName=P600; Kuka.BlendingEnabled=False; Kuka.MoveDataPtpName=PDAT1; Kuka.VelocityPtp=100; Kuka.VelocityFieldEnabled=True; Kuka.ColDetectFieldEnabled=True; Kuka.CurrentCDSetIndex=0; Kuka.MovementParameterFieldEnabled=True; IlfCommand=SPTP
        ;ENDFOLD
        SPTP XP600 WITH $VEL_AXIS[1] = SVEL_JOINT(100.0), $TOOL = STOOL2(FP600), $BASE = SBASE(FP600.BASE_NO), $IPO_MODE = SIPO_MODE(FP600.IPO_FRAME), $LOAD = SLOAD(FP600.TOOL_NO), $ACC_AXIS[1] = SACC_JOINT(PPDAT1), $APO = SAPO_PTP(PPDAT1), $GEAR_JERK[1] = SGEAR_JERK(PPDAT1), $COLLMON_TOL_PRO[1] = USE_CM_PRO_VALUES(0)
        ;ENDFOLD
        ;FOLD SLIN P601 Vel=0.1 m/s CPDAT27 Tool[1]:SMC Base[0] ;%{PE}
        ;FOLD Parameters ;%{h}
        ;Params IlfProvider=kukaroboter.basistech.inlineforms.movement.spline; Kuka.IsGlobalPoint=False; Kuka.PointName=P601; Kuka.BlendingEnabled=False; Kuka.MoveDataName=CPDAT27; Kuka.VelocityPath=0.1; Kuka.VelocityFieldEnabled=True; Kuka.ColDetectFieldEnabled=True; Kuka.CurrentCDSetIndex=0; Kuka.MovementParameterFieldEnabled=True; IlfCommand=SLIN
        ;ENDFOLD
        SLIN XP601 WITH $VEL = SVEL_CP(0.1, , LCPDAT27), $TOOL = STOOL2(FP601), $BASE = SBASE(FP601.BASE_NO), $IPO_MODE = SIPO_MODE(FP601.IPO_FRAME), $LOAD = SLOAD(FP601.TOOL_NO), $ACC = SACC_CP(LCPDAT27), $ORI_TYPE = SORI_TYP(LCPDAT27), $APO = SAPO(LCPDAT27), $JERK = SJERK(LCPDAT27), $COLLMON_TOL_PRO[1] = USE_CM_PRO_VALUES(0)
        ;ENDFOLD
        ;FOLD SLIN P602 Vel=0.1 m/s CPDAT27 Tool[1]:SMC Base[0] ;%{PE}
        ;FOLD Parameters ;%{h}
        ;Params IlfProvider=kukaroboter.basistech.inlineforms.movement.spline; Kuka.IsGlobalPoint=False; Kuka.PointName=P602; Kuka.BlendingEnabled=False; Kuka.MoveDataName=CPDAT27; Kuka.VelocityPath=0.1; Kuka.VelocityFieldEnabled=True; Kuka.ColDetectFieldEnabled=True; Kuka.CurrentCDSetIndex=0; Kuka.MovementParameterFieldEnabled=True; IlfCommand=SLIN
        ;ENDFOLD
        SLIN XP602 WITH $VEL = SVEL_CP(0.1, , LCPDAT27), $TOOL = STOOL2(FP602), $BASE = SBASE(FP602.BASE_NO), $IPO_MODE = SIPO_MODE(FP602.IPO_FRAME), $LOAD = SLOAD(FP602.TOOL_NO), $ACC = SACC_CP(LCPDAT27), $ORI_TYPE = SORI_TYP(LCPDAT27), $APO = SAPO(LCPDAT27), $JERK = SJERK(LCPDAT27), $COLLMON_TOL_PRO[1] = USE_CM_PRO_VALUES(0)
        ;ENDFOLD
      ENDIF

      IF finalPosition == 42 THEN
        ;FOLD SPTP P142 Vel=100 % PDAT1 Tool[1]:SMC Base[0] ;%{PE}
        ;FOLD Parameters ;%{h}
        ;Params IlfProvider=kukaroboter.basistech.inlineforms.movement.spline; Kuka.IsGlobalPoint=False; Kuka.PointName=P142; Kuka.BlendingEnabled=False; Kuka.MoveDataPtpName=PDAT1; Kuka.VelocityPtp=100; Kuka.VelocityFieldEnabled=True; Kuka.ColDetectFieldEnabled=True; Kuka.CurrentCDSetIndex=0; Kuka.MovementParameterFieldEnabled=True; IlfCommand=SPTP
        ;ENDFOLD
        SPTP XP142 WITH $VEL_AXIS[1] = SVEL_JOINT(100.0), $TOOL = STOOL2(FP142), $BASE = SBASE(FP142.BASE_NO), $IPO_MODE = SIPO_MODE(FP142.IPO_FRAME), $LOAD = SLOAD(FP142.TOOL_NO), $ACC_AXIS[1] = SACC_JOINT(PPDAT1), $APO = SAPO_PTP(PPDAT1), $GEAR_JERK[1] = SGEAR_JERK(PPDAT1), $COLLMON_TOL_PRO[1] = USE_CM_PRO_VALUES(0)
        ;ENDFOLD
        ;FOLD SLIN P242 Vel=0.1 m/s CPDAT27 Tool[1]:SMC Base[0] ;%{PE}
        ;FOLD Parameters ;%{h}
        ;Params IlfProvider=kukaroboter.basistech.inlineforms.movement.spline; Kuka.IsGlobalPoint=False; Kuka.PointName=P242; Kuka.BlendingEnabled=False; Kuka.MoveDataName=CPDAT27; Kuka.VelocityPath=0.1; Kuka.VelocityFieldEnabled=True; Kuka.ColDetectFieldEnabled=True; Kuka.CurrentCDSetIndex=0; Kuka.MovementParameterFieldEnabled=True; IlfCommand=SLIN
        ;ENDFOLD
        SLIN XP242 WITH $VEL = SVEL_CP(0.1, , LCPDAT27), $TOOL = STOOL2(FP242), $BASE = SBASE(FP242.BASE_NO), $IPO_MODE = SIPO_MODE(FP242.IPO_FRAME), $LOAD = SLOAD(FP242.TOOL_NO), $ACC = SACC_CP(LCPDAT27), $ORI_TYPE = SORI_TYP(LCPDAT27), $APO = SAPO(LCPDAT27), $JERK = SJERK(LCPDAT27), $COLLMON_TOL_PRO[1] = USE_CM_PRO_VALUES(0)
        ;ENDFOLD
        ;FOLD Gripper SET [1]Gripper1 State=[1]ABIERTA Wait 0.2[s] Check with Strategy 1 ;%{PE}
        ;FOLD Parameters Parameters ;%{h}
        ;Params IlfProvider=GripperTech.GripperSet;setgripper=1;setstate=1;setcont=nocont;waittime=0.2;errorstrategy=1
        ;ENDFOLD
        GRPg_SetStateAndCheck(1, 1, 0.2, 1)
        ;ENDFOLD
        ;FOLD SLIN P142 Vel=0.1 m/s CPDAT28 Tool[1]:SMC Base[0] ;%{PE}
        ;FOLD Parameters ;%{h}
        ;Params IlfProvider=kukaroboter.basistech.inlineforms.movement.spline; Kuka.IsGlobalPoint=False; Kuka.PointName=P142; Kuka.BlendingEnabled=False; Kuka.MoveDataName=CPDAT28; Kuka.VelocityPath=0.1; Kuka.VelocityFieldEnabled=True; Kuka.ColDetectFieldEnabled=True; Kuka.CurrentCDSetIndex=0; Kuka.MovementParameterFieldEnabled=True; IlfCommand=SLIN
        ;ENDFOLD
        SLIN XP142 WITH $VEL = SVEL_CP(0.1, , LCPDAT28), $TOOL = STOOL2(FP142), $BASE = SBASE(FP142.BASE_NO), $IPO_MODE = SIPO_MODE(FP142.IPO_FRAME), $LOAD = SLOAD(FP142.TOOL_NO), $ACC = SACC_CP(LCPDAT28), $ORI_TYPE = SORI_TYP(LCPDAT28), $APO = SAPO(LCPDAT28), $JERK = SJERK(LCPDAT28), $COLLMON_TOL_PRO[1] = USE_CM_PRO_VALUES(0)
        ;ENDFOLD
        ;FOLD SPTP P600 Vel=100 % PDAT1 Tool[1]:SMC Base[0] ;%{PE}
        ;FOLD Parameters ;%{h}
        ;Params IlfProvider=kukaroboter.basistech.inlineforms.movement.spline; Kuka.IsGlobalPoint=False; Kuka.PointName=P600; Kuka.BlendingEnabled=False; Kuka.MoveDataPtpName=PDAT1; Kuka.VelocityPtp=100; Kuka.VelocityFieldEnabled=True; Kuka.ColDetectFieldEnabled=True; Kuka.CurrentCDSetIndex=0; Kuka.MovementParameterFieldEnabled=True; IlfCommand=SPTP
        ;ENDFOLD
        SPTP XP600 WITH $VEL_AXIS[1] = SVEL_JOINT(100.0), $TOOL = STOOL2(FP600), $BASE = SBASE(FP600.BASE_NO), $IPO_MODE = SIPO_MODE(FP600.IPO_FRAME), $LOAD = SLOAD(FP600.TOOL_NO), $ACC_AXIS[1] = SACC_JOINT(PPDAT1), $APO = SAPO_PTP(PPDAT1), $GEAR_JERK[1] = SGEAR_JERK(PPDAT1), $COLLMON_TOL_PRO[1] = USE_CM_PRO_VALUES(0)
        ;ENDFOLD
        ;FOLD SLIN P601 Vel=0.1 m/s CPDAT27 Tool[1]:SMC Base[0] ;%{PE}
        ;FOLD Parameters ;%{h}
        ;Params IlfProvider=kukaroboter.basistech.inlineforms.movement.spline; Kuka.IsGlobalPoint=False; Kuka.PointName=P601; Kuka.BlendingEnabled=False; Kuka.MoveDataName=CPDAT27; Kuka.VelocityPath=0.1; Kuka.VelocityFieldEnabled=True; Kuka.ColDetectFieldEnabled=True; Kuka.CurrentCDSetIndex=0; Kuka.MovementParameterFieldEnabled=True; IlfCommand=SLIN
        ;ENDFOLD
        SLIN XP601 WITH $VEL = SVEL_CP(0.1, , LCPDAT27), $TOOL = STOOL2(FP601), $BASE = SBASE(FP601.BASE_NO), $IPO_MODE = SIPO_MODE(FP601.IPO_FRAME), $LOAD = SLOAD(FP601.TOOL_NO), $ACC = SACC_CP(LCPDAT27), $ORI_TYPE = SORI_TYP(LCPDAT27), $APO = SAPO(LCPDAT27), $JERK = SJERK(LCPDAT27), $COLLMON_TOL_PRO[1] = USE_CM_PRO_VALUES(0)
        ;ENDFOLD
        ;FOLD SLIN P602 Vel=0.1 m/s CPDAT27 Tool[1]:SMC Base[0] ;%{PE}
        ;FOLD Parameters ;%{h}
        ;Params IlfProvider=kukaroboter.basistech.inlineforms.movement.spline; Kuka.IsGlobalPoint=False; Kuka.PointName=P602; Kuka.BlendingEnabled=False; Kuka.MoveDataName=CPDAT27; Kuka.VelocityPath=0.1; Kuka.VelocityFieldEnabled=True; Kuka.ColDetectFieldEnabled=True; Kuka.CurrentCDSetIndex=0; Kuka.MovementParameterFieldEnabled=True; IlfCommand=SLIN
        ;ENDFOLD
        SLIN XP602 WITH $VEL = SVEL_CP(0.1, , LCPDAT27), $TOOL = STOOL2(FP602), $BASE = SBASE(FP602.BASE_NO), $IPO_MODE = SIPO_MODE(FP602.IPO_FRAME), $LOAD = SLOAD(FP602.TOOL_NO), $ACC = SACC_CP(LCPDAT27), $ORI_TYPE = SORI_TYP(LCPDAT27), $APO = SAPO(LCPDAT27), $JERK = SJERK(LCPDAT27), $COLLMON_TOL_PRO[1] = USE_CM_PRO_VALUES(0)
        ;ENDFOLD
      ENDIF

      IF finalPosition == 43 THEN
        ;FOLD SPTP P143 Vel=100 % PDAT1 Tool[1]:SMC Base[0] ;%{PE}
        ;FOLD Parameters ;%{h}
        ;Params IlfProvider=kukaroboter.basistech.inlineforms.movement.spline; Kuka.IsGlobalPoint=False; Kuka.PointName=P143; Kuka.BlendingEnabled=False; Kuka.MoveDataPtpName=PDAT1; Kuka.VelocityPtp=100; Kuka.VelocityFieldEnabled=True; Kuka.ColDetectFieldEnabled=True; Kuka.CurrentCDSetIndex=0; Kuka.MovementParameterFieldEnabled=True; IlfCommand=SPTP
        ;ENDFOLD
        SPTP XP143 WITH $VEL_AXIS[1] = SVEL_JOINT(100.0), $TOOL = STOOL2(FP143), $BASE = SBASE(FP143.BASE_NO), $IPO_MODE = SIPO_MODE(FP143.IPO_FRAME), $LOAD = SLOAD(FP143.TOOL_NO), $ACC_AXIS[1] = SACC_JOINT(PPDAT1), $APO = SAPO_PTP(PPDAT1), $GEAR_JERK[1] = SGEAR_JERK(PPDAT1), $COLLMON_TOL_PRO[1] = USE_CM_PRO_VALUES(0)
        ;ENDFOLD
        ;FOLD SLIN P243 Vel=0.1 m/s CPDAT27 Tool[1]:SMC Base[0] ;%{PE}
        ;FOLD Parameters ;%{h}
        ;Params IlfProvider=kukaroboter.basistech.inlineforms.movement.spline; Kuka.IsGlobalPoint=False; Kuka.PointName=P243; Kuka.BlendingEnabled=False; Kuka.MoveDataName=CPDAT27; Kuka.VelocityPath=0.1; Kuka.VelocityFieldEnabled=True; Kuka.ColDetectFieldEnabled=True; Kuka.CurrentCDSetIndex=0; Kuka.MovementParameterFieldEnabled=True; IlfCommand=SLIN
        ;ENDFOLD
        SLIN XP243 WITH $VEL = SVEL_CP(0.1, , LCPDAT27), $TOOL = STOOL2(FP243), $BASE = SBASE(FP243.BASE_NO), $IPO_MODE = SIPO_MODE(FP243.IPO_FRAME), $LOAD = SLOAD(FP243.TOOL_NO), $ACC = SACC_CP(LCPDAT27), $ORI_TYPE = SORI_TYP(LCPDAT27), $APO = SAPO(LCPDAT27), $JERK = SJERK(LCPDAT27), $COLLMON_TOL_PRO[1] = USE_CM_PRO_VALUES(0)
        ;ENDFOLD
        ;FOLD Gripper SET [1]Gripper1 State=[1]ABIERTA Wait 0.2[s] Check with Strategy 1 ;%{PE}
        ;FOLD Parameters Parameters ;%{h}
        ;Params IlfProvider=GripperTech.GripperSet;setgripper=1;setstate=1;setcont=nocont;waittime=0.2;errorstrategy=1
        ;ENDFOLD
        GRPg_SetStateAndCheck(1, 1, 0.2, 1)
        ;ENDFOLD
        ;FOLD SLIN P143 Vel=0.1 m/s CPDAT28 Tool[1]:SMC Base[0] ;%{PE}
        ;FOLD Parameters ;%{h}
        ;Params IlfProvider=kukaroboter.basistech.inlineforms.movement.spline; Kuka.IsGlobalPoint=False; Kuka.PointName=P143; Kuka.BlendingEnabled=False; Kuka.MoveDataName=CPDAT28; Kuka.VelocityPath=0.1; Kuka.VelocityFieldEnabled=True; Kuka.ColDetectFieldEnabled=True; Kuka.CurrentCDSetIndex=0; Kuka.MovementParameterFieldEnabled=True; IlfCommand=SLIN
        ;ENDFOLD
        SLIN XP143 WITH $VEL = SVEL_CP(0.1, , LCPDAT28), $TOOL = STOOL2(FP143), $BASE = SBASE(FP143.BASE_NO), $IPO_MODE = SIPO_MODE(FP143.IPO_FRAME), $LOAD = SLOAD(FP143.TOOL_NO), $ACC = SACC_CP(LCPDAT28), $ORI_TYPE = SORI_TYP(LCPDAT28), $APO = SAPO(LCPDAT28), $JERK = SJERK(LCPDAT28), $COLLMON_TOL_PRO[1] = USE_CM_PRO_VALUES(0)
        ;ENDFOLD
        ;FOLD SPTP P600 Vel=100 % PDAT1 Tool[1]:SMC Base[0] ;%{PE}
        ;FOLD Parameters ;%{h}
        ;Params IlfProvider=kukaroboter.basistech.inlineforms.movement.spline; Kuka.IsGlobalPoint=False; Kuka.PointName=P600; Kuka.BlendingEnabled=False; Kuka.MoveDataPtpName=PDAT1; Kuka.VelocityPtp=100; Kuka.VelocityFieldEnabled=True; Kuka.ColDetectFieldEnabled=True; Kuka.CurrentCDSetIndex=0; Kuka.MovementParameterFieldEnabled=True; IlfCommand=SPTP
        ;ENDFOLD
        SPTP XP600 WITH $VEL_AXIS[1] = SVEL_JOINT(100.0), $TOOL = STOOL2(FP600), $BASE = SBASE(FP600.BASE_NO), $IPO_MODE = SIPO_MODE(FP600.IPO_FRAME), $LOAD = SLOAD(FP600.TOOL_NO), $ACC_AXIS[1] = SACC_JOINT(PPDAT1), $APO = SAPO_PTP(PPDAT1), $GEAR_JERK[1] = SGEAR_JERK(PPDAT1), $COLLMON_TOL_PRO[1] = USE_CM_PRO_VALUES(0)
        ;ENDFOLD
        ;FOLD SLIN P601 Vel=0.1 m/s CPDAT27 Tool[1]:SMC Base[0] ;%{PE}
        ;FOLD Parameters ;%{h}
        ;Params IlfProvider=kukaroboter.basistech.inlineforms.movement.spline; Kuka.IsGlobalPoint=False; Kuka.PointName=P601; Kuka.BlendingEnabled=False; Kuka.MoveDataName=CPDAT27; Kuka.VelocityPath=0.1; Kuka.VelocityFieldEnabled=True; Kuka.ColDetectFieldEnabled=True; Kuka.CurrentCDSetIndex=0; Kuka.MovementParameterFieldEnabled=True; IlfCommand=SLIN
        ;ENDFOLD
        SLIN XP601 WITH $VEL = SVEL_CP(0.1, , LCPDAT27), $TOOL = STOOL2(FP601), $BASE = SBASE(FP601.BASE_NO), $IPO_MODE = SIPO_MODE(FP601.IPO_FRAME), $LOAD = SLOAD(FP601.TOOL_NO), $ACC = SACC_CP(LCPDAT27), $ORI_TYPE = SORI_TYP(LCPDAT27), $APO = SAPO(LCPDAT27), $JERK = SJERK(LCPDAT27), $COLLMON_TOL_PRO[1] = USE_CM_PRO_VALUES(0)
        ;ENDFOLD
        ;FOLD SLIN P602 Vel=0.1 m/s CPDAT27 Tool[1]:SMC Base[0] ;%{PE}
        ;FOLD Parameters ;%{h}
        ;Params IlfProvider=kukaroboter.basistech.inlineforms.movement.spline; Kuka.IsGlobalPoint=False; Kuka.PointName=P602; Kuka.BlendingEnabled=False; Kuka.MoveDataName=CPDAT27; Kuka.VelocityPath=0.1; Kuka.VelocityFieldEnabled=True; Kuka.ColDetectFieldEnabled=True; Kuka.CurrentCDSetIndex=0; Kuka.MovementParameterFieldEnabled=True; IlfCommand=SLIN
        ;ENDFOLD
        SLIN XP602 WITH $VEL = SVEL_CP(0.1, , LCPDAT27), $TOOL = STOOL2(FP602), $BASE = SBASE(FP602.BASE_NO), $IPO_MODE = SIPO_MODE(FP602.IPO_FRAME), $LOAD = SLOAD(FP602.TOOL_NO), $ACC = SACC_CP(LCPDAT27), $ORI_TYPE = SORI_TYP(LCPDAT27), $APO = SAPO(LCPDAT27), $JERK = SJERK(LCPDAT27), $COLLMON_TOL_PRO[1] = USE_CM_PRO_VALUES(0)
        ;ENDFOLD
      ENDIF

      IF finalPosition == 44 THEN
        ;FOLD SPTP P144 Vel=100 % PDAT1 Tool[1]:SMC Base[0] ;%{PE}
        ;FOLD Parameters ;%{h}
        ;Params IlfProvider=kukaroboter.basistech.inlineforms.movement.spline; Kuka.IsGlobalPoint=False; Kuka.PointName=P144; Kuka.BlendingEnabled=False; Kuka.MoveDataPtpName=PDAT1; Kuka.VelocityPtp=100; Kuka.VelocityFieldEnabled=True; Kuka.ColDetectFieldEnabled=True; Kuka.CurrentCDSetIndex=0; Kuka.MovementParameterFieldEnabled=True; IlfCommand=SPTP
        ;ENDFOLD
        SPTP XP144 WITH $VEL_AXIS[1] = SVEL_JOINT(100.0), $TOOL = STOOL2(FP144), $BASE = SBASE(FP144.BASE_NO), $IPO_MODE = SIPO_MODE(FP144.IPO_FRAME), $LOAD = SLOAD(FP144.TOOL_NO), $ACC_AXIS[1] = SACC_JOINT(PPDAT1), $APO = SAPO_PTP(PPDAT1), $GEAR_JERK[1] = SGEAR_JERK(PPDAT1), $COLLMON_TOL_PRO[1] = USE_CM_PRO_VALUES(0)
        ;ENDFOLD
        ;FOLD SLIN P244 Vel=0.1 m/s CPDAT27 Tool[1]:SMC Base[0] ;%{PE}
        ;FOLD Parameters ;%{h}
        ;Params IlfProvider=kukaroboter.basistech.inlineforms.movement.spline; Kuka.IsGlobalPoint=False; Kuka.PointName=P244; Kuka.BlendingEnabled=False; Kuka.MoveDataName=CPDAT27; Kuka.VelocityPath=0.1; Kuka.VelocityFieldEnabled=True; Kuka.ColDetectFieldEnabled=True; Kuka.CurrentCDSetIndex=0; Kuka.MovementParameterFieldEnabled=True; IlfCommand=SLIN
        ;ENDFOLD
        SLIN XP244 WITH $VEL = SVEL_CP(0.1, , LCPDAT27), $TOOL = STOOL2(FP244), $BASE = SBASE(FP244.BASE_NO), $IPO_MODE = SIPO_MODE(FP244.IPO_FRAME), $LOAD = SLOAD(FP244.TOOL_NO), $ACC = SACC_CP(LCPDAT27), $ORI_TYPE = SORI_TYP(LCPDAT27), $APO = SAPO(LCPDAT27), $JERK = SJERK(LCPDAT27), $COLLMON_TOL_PRO[1] = USE_CM_PRO_VALUES(0)
        ;ENDFOLD
        ;FOLD Gripper SET [1]Gripper1 State=[1]ABIERTA Wait 0.2[s] Check with Strategy 1 ;%{PE}
        ;FOLD Parameters Parameters ;%{h}
        ;Params IlfProvider=GripperTech.GripperSet;setgripper=1;setstate=1;setcont=nocont;waittime=0.2;errorstrategy=1
        ;ENDFOLD
        GRPg_SetStateAndCheck(1, 1, 0.2, 1)
        ;ENDFOLD
        ;FOLD SLIN P144 Vel=0.1 m/s CPDAT28 Tool[1]:SMC Base[0] ;%{PE}
        ;FOLD Parameters ;%{h}
        ;Params IlfProvider=kukaroboter.basistech.inlineforms.movement.spline; Kuka.IsGlobalPoint=False; Kuka.PointName=P144; Kuka.BlendingEnabled=False; Kuka.MoveDataName=CPDAT28; Kuka.VelocityPath=0.1; Kuka.VelocityFieldEnabled=True; Kuka.ColDetectFieldEnabled=True; Kuka.CurrentCDSetIndex=0; Kuka.MovementParameterFieldEnabled=True; IlfCommand=SLIN
        ;ENDFOLD
        SLIN XP144 WITH $VEL = SVEL_CP(0.1, , LCPDAT28), $TOOL = STOOL2(FP144), $BASE = SBASE(FP144.BASE_NO), $IPO_MODE = SIPO_MODE(FP144.IPO_FRAME), $LOAD = SLOAD(FP144.TOOL_NO), $ACC = SACC_CP(LCPDAT28), $ORI_TYPE = SORI_TYP(LCPDAT28), $APO = SAPO(LCPDAT28), $JERK = SJERK(LCPDAT28), $COLLMON_TOL_PRO[1] = USE_CM_PRO_VALUES(0)
        ;ENDFOLD
        ;FOLD SPTP P600 Vel=100 % PDAT1 Tool[1]:SMC Base[0] ;%{PE}
        ;FOLD Parameters ;%{h}
        ;Params IlfProvider=kukaroboter.basistech.inlineforms.movement.spline; Kuka.IsGlobalPoint=False; Kuka.PointName=P600; Kuka.BlendingEnabled=False; Kuka.MoveDataPtpName=PDAT1; Kuka.VelocityPtp=100; Kuka.VelocityFieldEnabled=True; Kuka.ColDetectFieldEnabled=True; Kuka.CurrentCDSetIndex=0; Kuka.MovementParameterFieldEnabled=True; IlfCommand=SPTP
        ;ENDFOLD
        SPTP XP600 WITH $VEL_AXIS[1] = SVEL_JOINT(100.0), $TOOL = STOOL2(FP600), $BASE = SBASE(FP600.BASE_NO), $IPO_MODE = SIPO_MODE(FP600.IPO_FRAME), $LOAD = SLOAD(FP600.TOOL_NO), $ACC_AXIS[1] = SACC_JOINT(PPDAT1), $APO = SAPO_PTP(PPDAT1), $GEAR_JERK[1] = SGEAR_JERK(PPDAT1), $COLLMON_TOL_PRO[1] = USE_CM_PRO_VALUES(0)
        ;ENDFOLD
        ;FOLD SLIN P601 Vel=0.1 m/s CPDAT27 Tool[1]:SMC Base[0] ;%{PE}
        ;FOLD Parameters ;%{h}
        ;Params IlfProvider=kukaroboter.basistech.inlineforms.movement.spline; Kuka.IsGlobalPoint=False; Kuka.PointName=P601; Kuka.BlendingEnabled=False; Kuka.MoveDataName=CPDAT27; Kuka.VelocityPath=0.1; Kuka.VelocityFieldEnabled=True; Kuka.ColDetectFieldEnabled=True; Kuka.CurrentCDSetIndex=0; Kuka.MovementParameterFieldEnabled=True; IlfCommand=SLIN
        ;ENDFOLD
        SLIN XP601 WITH $VEL = SVEL_CP(0.1, , LCPDAT27), $TOOL = STOOL2(FP601), $BASE = SBASE(FP601.BASE_NO), $IPO_MODE = SIPO_MODE(FP601.IPO_FRAME), $LOAD = SLOAD(FP601.TOOL_NO), $ACC = SACC_CP(LCPDAT27), $ORI_TYPE = SORI_TYP(LCPDAT27), $APO = SAPO(LCPDAT27), $JERK = SJERK(LCPDAT27), $COLLMON_TOL_PRO[1] = USE_CM_PRO_VALUES(0)
        ;ENDFOLD
        ;FOLD SLIN P602 Vel=0.1 m/s CPDAT27 Tool[1]:SMC Base[0] ;%{PE}
        ;FOLD Parameters ;%{h}
        ;Params IlfProvider=kukaroboter.basistech.inlineforms.movement.spline; Kuka.IsGlobalPoint=False; Kuka.PointName=P602; Kuka.BlendingEnabled=False; Kuka.MoveDataName=CPDAT27; Kuka.VelocityPath=0.1; Kuka.VelocityFieldEnabled=True; Kuka.ColDetectFieldEnabled=True; Kuka.CurrentCDSetIndex=0; Kuka.MovementParameterFieldEnabled=True; IlfCommand=SLIN
        ;ENDFOLD
        SLIN XP602 WITH $VEL = SVEL_CP(0.1, , LCPDAT27), $TOOL = STOOL2(FP602), $BASE = SBASE(FP602.BASE_NO), $IPO_MODE = SIPO_MODE(FP602.IPO_FRAME), $LOAD = SLOAD(FP602.TOOL_NO), $ACC = SACC_CP(LCPDAT27), $ORI_TYPE = SORI_TYP(LCPDAT27), $APO = SAPO(LCPDAT27), $JERK = SJERK(LCPDAT27), $COLLMON_TOL_PRO[1] = USE_CM_PRO_VALUES(0)
        ;ENDFOLD
      ENDIF

      IF finalPosition == 45 THEN
        ;FOLD SPTP P145 Vel=100 % PDAT1 Tool[1]:SMC Base[0] ;%{PE}
        ;FOLD Parameters ;%{h}
        ;Params IlfProvider=kukaroboter.basistech.inlineforms.movement.spline; Kuka.IsGlobalPoint=False; Kuka.PointName=P145; Kuka.BlendingEnabled=False; Kuka.MoveDataPtpName=PDAT1; Kuka.VelocityPtp=100; Kuka.VelocityFieldEnabled=True; Kuka.ColDetectFieldEnabled=True; Kuka.CurrentCDSetIndex=0; Kuka.MovementParameterFieldEnabled=True; IlfCommand=SPTP
        ;ENDFOLD
        SPTP XP145 WITH $VEL_AXIS[1] = SVEL_JOINT(100.0), $TOOL = STOOL2(FP145), $BASE = SBASE(FP145.BASE_NO), $IPO_MODE = SIPO_MODE(FP145.IPO_FRAME), $LOAD = SLOAD(FP145.TOOL_NO), $ACC_AXIS[1] = SACC_JOINT(PPDAT1), $APO = SAPO_PTP(PPDAT1), $GEAR_JERK[1] = SGEAR_JERK(PPDAT1), $COLLMON_TOL_PRO[1] = USE_CM_PRO_VALUES(0)
        ;ENDFOLD
        ;FOLD SLIN P245 Vel=0.1 m/s CPDAT27 Tool[1]:SMC Base[0] ;%{PE}
        ;FOLD Parameters ;%{h}
        ;Params IlfProvider=kukaroboter.basistech.inlineforms.movement.spline; Kuka.IsGlobalPoint=False; Kuka.PointName=P245; Kuka.BlendingEnabled=False; Kuka.MoveDataName=CPDAT27; Kuka.VelocityPath=0.1; Kuka.VelocityFieldEnabled=True; Kuka.ColDetectFieldEnabled=True; Kuka.CurrentCDSetIndex=0; Kuka.MovementParameterFieldEnabled=True; IlfCommand=SLIN
        ;ENDFOLD
        SLIN XP245 WITH $VEL = SVEL_CP(0.1, , LCPDAT27), $TOOL = STOOL2(FP245), $BASE = SBASE(FP245.BASE_NO), $IPO_MODE = SIPO_MODE(FP245.IPO_FRAME), $LOAD = SLOAD(FP245.TOOL_NO), $ACC = SACC_CP(LCPDAT27), $ORI_TYPE = SORI_TYP(LCPDAT27), $APO = SAPO(LCPDAT27), $JERK = SJERK(LCPDAT27), $COLLMON_TOL_PRO[1] = USE_CM_PRO_VALUES(0)
        ;ENDFOLD
        ;FOLD Gripper SET [1]Gripper1 State=[1]ABIERTA Wait 0.2[s] Check with Strategy 1 ;%{PE}
        ;FOLD Parameters Parameters ;%{h}
        ;Params IlfProvider=GripperTech.GripperSet;setgripper=1;setstate=1;setcont=nocont;waittime=0.2;errorstrategy=1
        ;ENDFOLD
        GRPg_SetStateAndCheck(1, 1, 0.2, 1)
        ;ENDFOLD
        ;FOLD SLIN P145 Vel=0.1 m/s CPDAT28 Tool[1]:SMC Base[0] ;%{PE}
        ;FOLD Parameters ;%{h}
        ;Params IlfProvider=kukaroboter.basistech.inlineforms.movement.spline; Kuka.IsGlobalPoint=False; Kuka.PointName=P145; Kuka.BlendingEnabled=False; Kuka.MoveDataName=CPDAT28; Kuka.VelocityPath=0.1; Kuka.VelocityFieldEnabled=True; Kuka.ColDetectFieldEnabled=True; Kuka.CurrentCDSetIndex=0; Kuka.MovementParameterFieldEnabled=True; IlfCommand=SLIN
        ;ENDFOLD
        SLIN XP145 WITH $VEL = SVEL_CP(0.1, , LCPDAT28), $TOOL = STOOL2(FP145), $BASE = SBASE(FP145.BASE_NO), $IPO_MODE = SIPO_MODE(FP145.IPO_FRAME), $LOAD = SLOAD(FP145.TOOL_NO), $ACC = SACC_CP(LCPDAT28), $ORI_TYPE = SORI_TYP(LCPDAT28), $APO = SAPO(LCPDAT28), $JERK = SJERK(LCPDAT28), $COLLMON_TOL_PRO[1] = USE_CM_PRO_VALUES(0)
        ;ENDFOLD
        ;FOLD SPTP P600 Vel=100 % PDAT1 Tool[1]:SMC Base[0] ;%{PE}
        ;FOLD Parameters ;%{h}
        ;Params IlfProvider=kukaroboter.basistech.inlineforms.movement.spline; Kuka.IsGlobalPoint=False; Kuka.PointName=P600; Kuka.BlendingEnabled=False; Kuka.MoveDataPtpName=PDAT1; Kuka.VelocityPtp=100; Kuka.VelocityFieldEnabled=True; Kuka.ColDetectFieldEnabled=True; Kuka.CurrentCDSetIndex=0; Kuka.MovementParameterFieldEnabled=True; IlfCommand=SPTP
        ;ENDFOLD
        SPTP XP600 WITH $VEL_AXIS[1] = SVEL_JOINT(100.0), $TOOL = STOOL2(FP600), $BASE = SBASE(FP600.BASE_NO), $IPO_MODE = SIPO_MODE(FP600.IPO_FRAME), $LOAD = SLOAD(FP600.TOOL_NO), $ACC_AXIS[1] = SACC_JOINT(PPDAT1), $APO = SAPO_PTP(PPDAT1), $GEAR_JERK[1] = SGEAR_JERK(PPDAT1), $COLLMON_TOL_PRO[1] = USE_CM_PRO_VALUES(0)
        ;ENDFOLD
        ;FOLD SLIN P601 Vel=0.1 m/s CPDAT27 Tool[1]:SMC Base[0] ;%{PE}
        ;FOLD Parameters ;%{h}
        ;Params IlfProvider=kukaroboter.basistech.inlineforms.movement.spline; Kuka.IsGlobalPoint=False; Kuka.PointName=P601; Kuka.BlendingEnabled=False; Kuka.MoveDataName=CPDAT27; Kuka.VelocityPath=0.1; Kuka.VelocityFieldEnabled=True; Kuka.ColDetectFieldEnabled=True; Kuka.CurrentCDSetIndex=0; Kuka.MovementParameterFieldEnabled=True; IlfCommand=SLIN
        ;ENDFOLD
        SLIN XP601 WITH $VEL = SVEL_CP(0.1, , LCPDAT27), $TOOL = STOOL2(FP601), $BASE = SBASE(FP601.BASE_NO), $IPO_MODE = SIPO_MODE(FP601.IPO_FRAME), $LOAD = SLOAD(FP601.TOOL_NO), $ACC = SACC_CP(LCPDAT27), $ORI_TYPE = SORI_TYP(LCPDAT27), $APO = SAPO(LCPDAT27), $JERK = SJERK(LCPDAT27), $COLLMON_TOL_PRO[1] = USE_CM_PRO_VALUES(0)
        ;ENDFOLD
        ;FOLD SLIN P602 Vel=0.1 m/s CPDAT27 Tool[1]:SMC Base[0] ;%{PE}
        ;FOLD Parameters ;%{h}
        ;Params IlfProvider=kukaroboter.basistech.inlineforms.movement.spline; Kuka.IsGlobalPoint=False; Kuka.PointName=P602; Kuka.BlendingEnabled=False; Kuka.MoveDataName=CPDAT27; Kuka.VelocityPath=0.1; Kuka.VelocityFieldEnabled=True; Kuka.ColDetectFieldEnabled=True; Kuka.CurrentCDSetIndex=0; Kuka.MovementParameterFieldEnabled=True; IlfCommand=SLIN
        ;ENDFOLD
        SLIN XP602 WITH $VEL = SVEL_CP(0.1, , LCPDAT27), $TOOL = STOOL2(FP602), $BASE = SBASE(FP602.BASE_NO), $IPO_MODE = SIPO_MODE(FP602.IPO_FRAME), $LOAD = SLOAD(FP602.TOOL_NO), $ACC = SACC_CP(LCPDAT27), $ORI_TYPE = SORI_TYP(LCPDAT27), $APO = SAPO(LCPDAT27), $JERK = SJERK(LCPDAT27), $COLLMON_TOL_PRO[1] = USE_CM_PRO_VALUES(0)
        ;ENDFOLD
      ENDIF

      IF finalPosition == 46 THEN
        ;FOLD SPTP P146 Vel=100 % PDAT1 Tool[1]:SMC Base[0] ;%{PE}
        ;FOLD Parameters ;%{h}
        ;Params IlfProvider=kukaroboter.basistech.inlineforms.movement.spline; Kuka.IsGlobalPoint=False; Kuka.PointName=P146; Kuka.BlendingEnabled=False; Kuka.MoveDataPtpName=PDAT1; Kuka.VelocityPtp=100; Kuka.VelocityFieldEnabled=True; Kuka.ColDetectFieldEnabled=True; Kuka.CurrentCDSetIndex=0; Kuka.MovementParameterFieldEnabled=True; IlfCommand=SPTP
        ;ENDFOLD
        SPTP XP146 WITH $VEL_AXIS[1] = SVEL_JOINT(100.0), $TOOL = STOOL2(FP146), $BASE = SBASE(FP146.BASE_NO), $IPO_MODE = SIPO_MODE(FP146.IPO_FRAME), $LOAD = SLOAD(FP146.TOOL_NO), $ACC_AXIS[1] = SACC_JOINT(PPDAT1), $APO = SAPO_PTP(PPDAT1), $GEAR_JERK[1] = SGEAR_JERK(PPDAT1), $COLLMON_TOL_PRO[1] = USE_CM_PRO_VALUES(0)
        ;ENDFOLD
        ;FOLD SLIN P246 Vel=0.1 m/s CPDAT27 Tool[1]:SMC Base[0] ;%{PE}
        ;FOLD Parameters ;%{h}
        ;Params IlfProvider=kukaroboter.basistech.inlineforms.movement.spline; Kuka.IsGlobalPoint=False; Kuka.PointName=P246; Kuka.BlendingEnabled=False; Kuka.MoveDataName=CPDAT27; Kuka.VelocityPath=0.1; Kuka.VelocityFieldEnabled=True; Kuka.ColDetectFieldEnabled=True; Kuka.CurrentCDSetIndex=0; Kuka.MovementParameterFieldEnabled=True; IlfCommand=SLIN
        ;ENDFOLD
        SLIN XP246 WITH $VEL = SVEL_CP(0.1, , LCPDAT27), $TOOL = STOOL2(FP246), $BASE = SBASE(FP246.BASE_NO), $IPO_MODE = SIPO_MODE(FP246.IPO_FRAME), $LOAD = SLOAD(FP246.TOOL_NO), $ACC = SACC_CP(LCPDAT27), $ORI_TYPE = SORI_TYP(LCPDAT27), $APO = SAPO(LCPDAT27), $JERK = SJERK(LCPDAT27), $COLLMON_TOL_PRO[1] = USE_CM_PRO_VALUES(0)
        ;ENDFOLD
        ;FOLD Gripper SET [1]Gripper1 State=[1]ABIERTA Wait 0.2[s] Check with Strategy 1 ;%{PE}
        ;FOLD Parameters Parameters ;%{h}
        ;Params IlfProvider=GripperTech.GripperSet;setgripper=1;setstate=1;setcont=nocont;waittime=0.2;errorstrategy=1
        ;ENDFOLD
        GRPg_SetStateAndCheck(1, 1, 0.2, 1)
        ;ENDFOLD
        ;FOLD SLIN P146 Vel=0.1 m/s CPDAT28 Tool[1]:SMC Base[0] ;%{PE}
        ;FOLD Parameters ;%{h}
        ;Params IlfProvider=kukaroboter.basistech.inlineforms.movement.spline; Kuka.IsGlobalPoint=False; Kuka.PointName=P146; Kuka.BlendingEnabled=False; Kuka.MoveDataName=CPDAT28; Kuka.VelocityPath=0.1; Kuka.VelocityFieldEnabled=True; Kuka.ColDetectFieldEnabled=True; Kuka.CurrentCDSetIndex=0; Kuka.MovementParameterFieldEnabled=True; IlfCommand=SLIN
        ;ENDFOLD
        SLIN XP146 WITH $VEL = SVEL_CP(0.1, , LCPDAT28), $TOOL = STOOL2(FP146), $BASE = SBASE(FP146.BASE_NO), $IPO_MODE = SIPO_MODE(FP146.IPO_FRAME), $LOAD = SLOAD(FP146.TOOL_NO), $ACC = SACC_CP(LCPDAT28), $ORI_TYPE = SORI_TYP(LCPDAT28), $APO = SAPO(LCPDAT28), $JERK = SJERK(LCPDAT28), $COLLMON_TOL_PRO[1] = USE_CM_PRO_VALUES(0)
        ;ENDFOLD
        ;FOLD SPTP P600 Vel=100 % PDAT1 Tool[1]:SMC Base[0] ;%{PE}
        ;FOLD Parameters ;%{h}
        ;Params IlfProvider=kukaroboter.basistech.inlineforms.movement.spline; Kuka.IsGlobalPoint=False; Kuka.PointName=P600; Kuka.BlendingEnabled=False; Kuka.MoveDataPtpName=PDAT1; Kuka.VelocityPtp=100; Kuka.VelocityFieldEnabled=True; Kuka.ColDetectFieldEnabled=True; Kuka.CurrentCDSetIndex=0; Kuka.MovementParameterFieldEnabled=True; IlfCommand=SPTP
        ;ENDFOLD
        SPTP XP600 WITH $VEL_AXIS[1] = SVEL_JOINT(100.0), $TOOL = STOOL2(FP600), $BASE = SBASE(FP600.BASE_NO), $IPO_MODE = SIPO_MODE(FP600.IPO_FRAME), $LOAD = SLOAD(FP600.TOOL_NO), $ACC_AXIS[1] = SACC_JOINT(PPDAT1), $APO = SAPO_PTP(PPDAT1), $GEAR_JERK[1] = SGEAR_JERK(PPDAT1), $COLLMON_TOL_PRO[1] = USE_CM_PRO_VALUES(0)
        ;ENDFOLD
        ;FOLD SLIN P601 Vel=0.1 m/s CPDAT27 Tool[1]:SMC Base[0] ;%{PE}
        ;FOLD Parameters ;%{h}
        ;Params IlfProvider=kukaroboter.basistech.inlineforms.movement.spline; Kuka.IsGlobalPoint=False; Kuka.PointName=P601; Kuka.BlendingEnabled=False; Kuka.MoveDataName=CPDAT27; Kuka.VelocityPath=0.1; Kuka.VelocityFieldEnabled=True; Kuka.ColDetectFieldEnabled=True; Kuka.CurrentCDSetIndex=0; Kuka.MovementParameterFieldEnabled=True; IlfCommand=SLIN
        ;ENDFOLD
        SLIN XP601 WITH $VEL = SVEL_CP(0.1, , LCPDAT27), $TOOL = STOOL2(FP601), $BASE = SBASE(FP601.BASE_NO), $IPO_MODE = SIPO_MODE(FP601.IPO_FRAME), $LOAD = SLOAD(FP601.TOOL_NO), $ACC = SACC_CP(LCPDAT27), $ORI_TYPE = SORI_TYP(LCPDAT27), $APO = SAPO(LCPDAT27), $JERK = SJERK(LCPDAT27), $COLLMON_TOL_PRO[1] = USE_CM_PRO_VALUES(0)
        ;ENDFOLD
        ;FOLD SLIN P602 Vel=0.1 m/s CPDAT27 Tool[1]:SMC Base[0] ;%{PE}
        ;FOLD Parameters ;%{h}
        ;Params IlfProvider=kukaroboter.basistech.inlineforms.movement.spline; Kuka.IsGlobalPoint=False; Kuka.PointName=P602; Kuka.BlendingEnabled=False; Kuka.MoveDataName=CPDAT27; Kuka.VelocityPath=0.1; Kuka.VelocityFieldEnabled=True; Kuka.ColDetectFieldEnabled=True; Kuka.CurrentCDSetIndex=0; Kuka.MovementParameterFieldEnabled=True; IlfCommand=SLIN
        ;ENDFOLD
        SLIN XP602 WITH $VEL = SVEL_CP(0.1, , LCPDAT27), $TOOL = STOOL2(FP602), $BASE = SBASE(FP602.BASE_NO), $IPO_MODE = SIPO_MODE(FP602.IPO_FRAME), $LOAD = SLOAD(FP602.TOOL_NO), $ACC = SACC_CP(LCPDAT27), $ORI_TYPE = SORI_TYP(LCPDAT27), $APO = SAPO(LCPDAT27), $JERK = SJERK(LCPDAT27), $COLLMON_TOL_PRO[1] = USE_CM_PRO_VALUES(0)
        ;ENDFOLD
      ENDIF

      IF finalPosition == 47 THEN
        ;FOLD SPTP P147 Vel=100 % PDAT1 Tool[1]:SMC Base[0] ;%{PE}
        ;FOLD Parameters ;%{h}
        ;Params IlfProvider=kukaroboter.basistech.inlineforms.movement.spline; Kuka.IsGlobalPoint=False; Kuka.PointName=P147; Kuka.BlendingEnabled=False; Kuka.MoveDataPtpName=PDAT1; Kuka.VelocityPtp=100; Kuka.VelocityFieldEnabled=True; Kuka.ColDetectFieldEnabled=True; Kuka.CurrentCDSetIndex=0; Kuka.MovementParameterFieldEnabled=True; IlfCommand=SPTP
        ;ENDFOLD
        SPTP XP147 WITH $VEL_AXIS[1] = SVEL_JOINT(100.0), $TOOL = STOOL2(FP147), $BASE = SBASE(FP147.BASE_NO), $IPO_MODE = SIPO_MODE(FP147.IPO_FRAME), $LOAD = SLOAD(FP147.TOOL_NO), $ACC_AXIS[1] = SACC_JOINT(PPDAT1), $APO = SAPO_PTP(PPDAT1), $GEAR_JERK[1] = SGEAR_JERK(PPDAT1), $COLLMON_TOL_PRO[1] = USE_CM_PRO_VALUES(0)
        ;ENDFOLD
        ;FOLD SLIN P247 Vel=0.1 m/s CPDAT27 Tool[1]:SMC Base[0] ;%{PE}
        ;FOLD Parameters ;%{h}
        ;Params IlfProvider=kukaroboter.basistech.inlineforms.movement.spline; Kuka.IsGlobalPoint=False; Kuka.PointName=P247; Kuka.BlendingEnabled=False; Kuka.MoveDataName=CPDAT27; Kuka.VelocityPath=0.1; Kuka.VelocityFieldEnabled=True; Kuka.ColDetectFieldEnabled=True; Kuka.CurrentCDSetIndex=0; Kuka.MovementParameterFieldEnabled=True; IlfCommand=SLIN
        ;ENDFOLD
        SLIN XP247 WITH $VEL = SVEL_CP(0.1, , LCPDAT27), $TOOL = STOOL2(FP247), $BASE = SBASE(FP247.BASE_NO), $IPO_MODE = SIPO_MODE(FP247.IPO_FRAME), $LOAD = SLOAD(FP247.TOOL_NO), $ACC = SACC_CP(LCPDAT27), $ORI_TYPE = SORI_TYP(LCPDAT27), $APO = SAPO(LCPDAT27), $JERK = SJERK(LCPDAT27), $COLLMON_TOL_PRO[1] = USE_CM_PRO_VALUES(0)
        ;ENDFOLD
        ;FOLD Gripper SET [1]Gripper1 State=[1]ABIERTA Wait 0.2[s] Check with Strategy 1 ;%{PE}
        ;FOLD Parameters Parameters ;%{h}
        ;Params IlfProvider=GripperTech.GripperSet;setgripper=1;setstate=1;setcont=nocont;waittime=0.2;errorstrategy=1
        ;ENDFOLD
        GRPg_SetStateAndCheck(1, 1, 0.2, 1)
        ;ENDFOLD
        ;FOLD SLIN P147 Vel=0.1 m/s CPDAT28 Tool[1]:SMC Base[0] ;%{PE}
        ;FOLD Parameters ;%{h}
        ;Params IlfProvider=kukaroboter.basistech.inlineforms.movement.spline; Kuka.IsGlobalPoint=False; Kuka.PointName=P147; Kuka.BlendingEnabled=False; Kuka.MoveDataName=CPDAT28; Kuka.VelocityPath=0.1; Kuka.VelocityFieldEnabled=True; Kuka.ColDetectFieldEnabled=True; Kuka.CurrentCDSetIndex=0; Kuka.MovementParameterFieldEnabled=True; IlfCommand=SLIN
        ;ENDFOLD
        SLIN XP147 WITH $VEL = SVEL_CP(0.1, , LCPDAT28), $TOOL = STOOL2(FP147), $BASE = SBASE(FP147.BASE_NO), $IPO_MODE = SIPO_MODE(FP147.IPO_FRAME), $LOAD = SLOAD(FP147.TOOL_NO), $ACC = SACC_CP(LCPDAT28), $ORI_TYPE = SORI_TYP(LCPDAT28), $APO = SAPO(LCPDAT28), $JERK = SJERK(LCPDAT28), $COLLMON_TOL_PRO[1] = USE_CM_PRO_VALUES(0)
        ;ENDFOLD
        ;FOLD SPTP P600 Vel=100 % PDAT1 Tool[1]:SMC Base[0] ;%{PE}
        ;FOLD Parameters ;%{h}
        ;Params IlfProvider=kukaroboter.basistech.inlineforms.movement.spline; Kuka.IsGlobalPoint=False; Kuka.PointName=P600; Kuka.BlendingEnabled=False; Kuka.MoveDataPtpName=PDAT1; Kuka.VelocityPtp=100; Kuka.VelocityFieldEnabled=True; Kuka.ColDetectFieldEnabled=True; Kuka.CurrentCDSetIndex=0; Kuka.MovementParameterFieldEnabled=True; IlfCommand=SPTP
        ;ENDFOLD
        SPTP XP600 WITH $VEL_AXIS[1] = SVEL_JOINT(100.0), $TOOL = STOOL2(FP600), $BASE = SBASE(FP600.BASE_NO), $IPO_MODE = SIPO_MODE(FP600.IPO_FRAME), $LOAD = SLOAD(FP600.TOOL_NO), $ACC_AXIS[1] = SACC_JOINT(PPDAT1), $APO = SAPO_PTP(PPDAT1), $GEAR_JERK[1] = SGEAR_JERK(PPDAT1), $COLLMON_TOL_PRO[1] = USE_CM_PRO_VALUES(0)
        ;ENDFOLD
        ;FOLD SLIN P601 Vel=0.1 m/s CPDAT27 Tool[1]:SMC Base[0] ;%{PE}
        ;FOLD Parameters ;%{h}
        ;Params IlfProvider=kukaroboter.basistech.inlineforms.movement.spline; Kuka.IsGlobalPoint=False; Kuka.PointName=P601; Kuka.BlendingEnabled=False; Kuka.MoveDataName=CPDAT27; Kuka.VelocityPath=0.1; Kuka.VelocityFieldEnabled=True; Kuka.ColDetectFieldEnabled=True; Kuka.CurrentCDSetIndex=0; Kuka.MovementParameterFieldEnabled=True; IlfCommand=SLIN
        ;ENDFOLD
        SLIN XP601 WITH $VEL = SVEL_CP(0.1, , LCPDAT27), $TOOL = STOOL2(FP601), $BASE = SBASE(FP601.BASE_NO), $IPO_MODE = SIPO_MODE(FP601.IPO_FRAME), $LOAD = SLOAD(FP601.TOOL_NO), $ACC = SACC_CP(LCPDAT27), $ORI_TYPE = SORI_TYP(LCPDAT27), $APO = SAPO(LCPDAT27), $JERK = SJERK(LCPDAT27), $COLLMON_TOL_PRO[1] = USE_CM_PRO_VALUES(0)
        ;ENDFOLD
        ;FOLD SLIN P602 Vel=0.1 m/s CPDAT27 Tool[1]:SMC Base[0] ;%{PE}
        ;FOLD Parameters ;%{h}
        ;Params IlfProvider=kukaroboter.basistech.inlineforms.movement.spline; Kuka.IsGlobalPoint=False; Kuka.PointName=P602; Kuka.BlendingEnabled=False; Kuka.MoveDataName=CPDAT27; Kuka.VelocityPath=0.1; Kuka.VelocityFieldEnabled=True; Kuka.ColDetectFieldEnabled=True; Kuka.CurrentCDSetIndex=0; Kuka.MovementParameterFieldEnabled=True; IlfCommand=SLIN
        ;ENDFOLD
        SLIN XP602 WITH $VEL = SVEL_CP(0.1, , LCPDAT27), $TOOL = STOOL2(FP602), $BASE = SBASE(FP602.BASE_NO), $IPO_MODE = SIPO_MODE(FP602.IPO_FRAME), $LOAD = SLOAD(FP602.TOOL_NO), $ACC = SACC_CP(LCPDAT27), $ORI_TYPE = SORI_TYP(LCPDAT27), $APO = SAPO(LCPDAT27), $JERK = SJERK(LCPDAT27), $COLLMON_TOL_PRO[1] = USE_CM_PRO_VALUES(0)
        ;ENDFOLD
      ENDIF

